//   Motion/Motion Instance <-> CX2020 (EtherCAT)/Term 1 (EK1200)/Term 2 (EK1122)/Rack#2B-01 Coupler (EK1100)/Rack#2B-09 ENC_RxG_XG (EL5042)
//     PlcTask Inputs/GVL_Main.M10.nRawEncoderULINT <-> FB Inputs Channel 1 compact/Position
//     PlcTask Inputs/GVL_Main.M11.nRawEncoderULINT <-> FB Inputs Channel 2/Position
//   Motion/Motion Instance <-> CX2020 (EtherCAT)/Term 1 (EK1200)/Term 2 (EK1122)/Rack#2B-01 Coupler (EK1100)/Rack#2B-10 ENC_YG1_YG2 (EL5042)
//     PlcTask Inputs/GVL_Main.M7.nRawEncoderULINT <-> FB Inputs Channel 1/Position
//     PlcTask Inputs/GVL_Main.M8.nRawEncoderULINT <-> FB Inputs Channel 2/Position
//   Motion/Motion Instance <-> CX2020 (EtherCAT)/Term 1 (EK1200)/Term 2 (EK1122)/Rack#2B-01 Coupler (EK1100)/Rack#2B-11 ENC_YG3_X1PM (EL5042)
//     PlcTask Inputs/GVL_Main.M12.nRawEncoderULINT <-> FB Inputs Channel 2/Position
//     PlcTask Inputs/GVL_Main.M9.nRawEncoderULINT <-> FB Inputs Channel 1/Position
//   Motion/Motion Instance <-> CX2020 (EtherCAT)/Term 1 (EK1200)/Term 2 (EK1122)/Rack#2B-01 Coupler (EK1100)/Rack#2B-12 ENC_X2PM_RzPM (EL5042)
//     PlcTask Inputs/GVL_Main.M13.nRawEncoderULINT <-> FB Inputs Channel 1/Position
//     PlcTask Inputs/GVL_Main.M14.nRawEncoderULINT <-> FB Inputs Channel 2/Position
//   Motion/Motion Instance <-> CX2020 (EtherCAT)/Term 1 (EK1200)/Term 2 (EK1122)/Rack#2B-01 Coupler (EK1100)/Rack#2B-15 DR_YDF1 (EL7041-0052)
//     PlcTask Inputs/GVL_Main.M15.bLimitBackwardEnable <-> STM Status/Status/Digital input 2
//     PlcTask Inputs/GVL_Main.M15.bLimitForwardEnable <-> STM Status/Status/Digital input 1
//   Motion/Motion Instance <-> CX2020 (EtherCAT)/Term 1 (EK1200)/Term 2 (EK1122)/Rack#2B-01 Coupler (EK1100)/Rack#2B-16 DR_YDF2 (EL7041-0052)
//     PlcTask Inputs/GVL_Main.M16.bLimitBackwardEnable <-> STM Status/Status/Digital input 2
//     PlcTask Inputs/GVL_Main.M16.bLimitForwardEnable <-> STM Status/Status/Digital input 1
//   Motion/Motion Instance <-> CX2020 (EtherCAT)/Term 1 (EK1200)/Term 2 (EK1122)/Rack#2B-01 Coupler (EK1100)/Rack#2B-18 MB_ZF (EL2602)
//     PlcTask Outputs/GVL_Main.M27.bBrakeRelease <-> Channel 1/Output
//   Motion/Motion Instance <-> CX2020 (EtherCAT)/Term 1 (EK1200)/Term 2 (EK1122)/Rack#2B-01 Coupler (EK1100)/Rack#2B-19 DR_YDF3 (EL7041-0052)
//     PlcTask Inputs/GVL_Main.M17.bLimitBackwardEnable <-> STM Status/Status/Digital input 2
//     PlcTask Inputs/GVL_Main.M17.bLimitForwardEnable <-> STM Status/Status/Digital input 1
//   Motion/Motion Instance <-> CX2020 (EtherCAT)/Term 1 (EK1200)/Term 2 (EK1122)/Rack#2D LinearGaugeAmp (SC-HG1-ETC)
//     PlcTask Inputs/GVL_Sensor.stHDF.iRawCnts <-> Process Data(In)  TxPDO-Map/Response Data Unit4
//     PlcTask Inputs/GVL_Sensor.stYDF1.iRawCnts <-> Process Data(In)  TxPDO-Map/Response Data Unit1
//     PlcTask Inputs/GVL_Sensor.stYDF2.iRawCnts <-> Process Data(In)  TxPDO-Map/Response Data Unit2
//     PlcTask Inputs/GVL_Sensor.stYDF3.iRawCnts <-> Process Data(In)  TxPDO-Map/Response Data Unit3
//     PlcTask Outputs/PRG_Sensor.bSensorHeadNormalValueMode <-> Process Data(Out) RxPDO-Map/Normal Value Mode
//     PlcTask Outputs/PRG_Sensor.bSensorHeadValueMode <-> Process Data(Out) RxPDO-Map/Head Value Mode
//   Motion/Motion Instance <-> NC-Task 1 SAF/Axes/RxG
//     PlcTask Inputs/GVL_Main.M10.Axis.NcToPlc <-> Outputs/ToPlc
//     PlcTask Outputs/GVL_Main.M10.Axis.PlcToNc <-> Inputs/FromPlc
//   Motion/Motion Instance <-> NC-Task 1 SAF/Axes/RyDC
//     PlcTask Inputs/GVL_Main.M23.Axis.NcToPlc <-> Outputs/ToPlc
//     PlcTask Outputs/GVL_Main.M23.Axis.PlcToNc <-> Inputs/FromPlc
//   Motion/Motion Instance <-> NC-Task 1 SAF/Axes/RzPM
//     PlcTask Inputs/GVL_Main.M14.Axis.NcToPlc <-> Outputs/ToPlc
//     PlcTask Outputs/GVL_Main.M14.Axis.PlcToNc <-> Inputs/FromPlc
//   Motion/Motion Instance <-> NC-Task 1 SAF/Axes/Stepper
//     PlcTask Inputs/GVL_Main.M2.Axis.NcToPlc <-> Outputs/ToPlc
//     PlcTask Outputs/GVL_Main.M2.Axis.PlcToNc <-> Inputs/FromPlc
//   Motion/Motion Instance <-> NC-Task 1 SAF/Axes/XDC
//     PlcTask Inputs/GVL_Main.M22.Axis.NcToPlc <-> Outputs/ToPlc
//     PlcTask Outputs/GVL_Main.M22.Axis.PlcToNc <-> Inputs/FromPlc
//   Motion/Motion Instance <-> NC-Task 1 SAF/Axes/XG
//     PlcTask Inputs/GVL_Main.M11.Axis.NcToPlc <-> Outputs/ToPlc
//     PlcTask Outputs/GVL_Main.M11.Axis.PlcToNc <-> Inputs/FromPlc
//   Motion/Motion Instance <-> NC-Task 1 SAF/Axes/XPM1
//     PlcTask Inputs/GVL_Main.M12.Axis.NcToPlc <-> Outputs/ToPlc
//     PlcTask Outputs/GVL_Main.M12.Axis.PlcToNc <-> Inputs/FromPlc
//   Motion/Motion Instance <-> NC-Task 1 SAF/Axes/XPM2
//     PlcTask Inputs/GVL_Main.M13.Axis.NcToPlc <-> Outputs/ToPlc
//     PlcTask Outputs/GVL_Main.M13.Axis.PlcToNc <-> Inputs/FromPlc
//   Motion/Motion Instance <-> NC-Task 1 SAF/Axes/XS1
//     PlcTask Inputs/GVL_Main.M3.Axis.NcToPlc <-> Outputs/ToPlc
//     PlcTask Outputs/GVL_Main.M3.Axis.PlcToNc <-> Inputs/FromPlc
//   Motion/Motion Instance <-> NC-Task 1 SAF/Axes/XS2
//     PlcTask Inputs/GVL_Main.M4.Axis.NcToPlc <-> Outputs/ToPlc
//     PlcTask Outputs/GVL_Main.M4.Axis.PlcToNc <-> Inputs/FromPlc
//   Motion/Motion Instance <-> NC-Task 1 SAF/Axes/XSDC1
//     PlcTask Inputs/GVL_Main.M18.Axis.NcToPlc <-> Outputs/ToPlc
//     PlcTask Outputs/GVL_Main.M18.Axis.PlcToNc <-> Inputs/FromPlc
//   Motion/Motion Instance <-> NC-Task 1 SAF/Axes/XSDC2
//     PlcTask Inputs/GVL_Main.M19.Axis.NcToPlc <-> Outputs/ToPlc
//     PlcTask Outputs/GVL_Main.M19.Axis.PlcToNc <-> Inputs/FromPlc
//   Motion/Motion Instance <-> NC-Task 1 SAF/Axes/YDF1
//     PlcTask Inputs/GVL_Main.M15.Axis.NcToPlc <-> Outputs/ToPlc
//     PlcTask Outputs/GVL_Main.M15.Axis.PlcToNc <-> Inputs/FromPlc
//   Motion/Motion Instance <-> NC-Task 1 SAF/Axes/YDF2
//     PlcTask Inputs/GVL_Main.M16.Axis.NcToPlc <-> Outputs/ToPlc
//     PlcTask Outputs/GVL_Main.M16.Axis.PlcToNc <-> Inputs/FromPlc
//   Motion/Motion Instance <-> NC-Task 1 SAF/Axes/YDF3
//     PlcTask Inputs/GVL_Main.M17.Axis.NcToPlc <-> Outputs/ToPlc
//     PlcTask Outputs/GVL_Main.M17.Axis.PlcToNc <-> Inputs/FromPlc
//   Motion/Motion Instance <-> NC-Task 1 SAF/Axes/YF1
//     PlcTask Inputs/GVL_Main.M25.Axis.NcToPlc <-> Outputs/ToPlc
//     PlcTask Outputs/GVL_Main.M25.Axis.PlcToNc <-> Inputs/FromPlc
//   Motion/Motion Instance <-> NC-Task 1 SAF/Axes/YF2
//     PlcTask Inputs/GVL_Main.M26.Axis.NcToPlc <-> Outputs/ToPlc
//     PlcTask Outputs/GVL_Main.M26.Axis.PlcToNc <-> Inputs/FromPlc
//   Motion/Motion Instance <-> NC-Task 1 SAF/Axes/YG1
//     PlcTask Inputs/GVL_Main.M7.Axis.NcToPlc <-> Outputs/ToPlc
//     PlcTask Outputs/GVL_Main.M7.Axis.PlcToNc <-> Inputs/FromPlc
//   Motion/Motion Instance <-> NC-Task 1 SAF/Axes/YG2
//     PlcTask Inputs/GVL_Main.M8.Axis.NcToPlc <-> Outputs/ToPlc
//     PlcTask Outputs/GVL_Main.M8.Axis.PlcToNc <-> Inputs/FromPlc
//   Motion/Motion Instance <-> NC-Task 1 SAF/Axes/YG3
//     PlcTask Inputs/GVL_Main.M9.Axis.NcToPlc <-> Outputs/ToPlc
//     PlcTask Outputs/GVL_Main.M9.Axis.PlcToNc <-> Inputs/FromPlc
//   Motion/Motion Instance <-> NC-Task 1 SAF/Axes/YS1
//     PlcTask Inputs/GVL_Main.M5.Axis.NcToPlc <-> Outputs/ToPlc
//     PlcTask Outputs/GVL_Main.M5.Axis.PlcToNc <-> Inputs/FromPlc
//   Motion/Motion Instance <-> NC-Task 1 SAF/Axes/YS2
//     PlcTask Inputs/GVL_Main.M6.Axis.NcToPlc <-> Outputs/ToPlc
//     PlcTask Outputs/GVL_Main.M6.Axis.PlcToNc <-> Inputs/FromPlc
//   Motion/Motion Instance <-> NC-Task 1 SAF/Axes/YSDC1
//     PlcTask Inputs/GVL_Main.M20.Axis.NcToPlc <-> Outputs/ToPlc
//     PlcTask Outputs/GVL_Main.M20.Axis.PlcToNc <-> Inputs/FromPlc
//   Motion/Motion Instance <-> NC-Task 1 SAF/Axes/YSDC2
//     PlcTask Inputs/GVL_Main.M21.Axis.NcToPlc <-> Outputs/ToPlc
//     PlcTask Outputs/GVL_Main.M21.Axis.PlcToNc <-> Inputs/FromPlc
//   Motion/Motion Instance <-> NC-Task 1 SAF/Axes/ZDC
//     PlcTask Inputs/GVL_Main.M24.Axis.NcToPlc <-> Outputs/ToPlc
//     PlcTask Outputs/GVL_Main.M24.Axis.PlcToNc <-> Inputs/FromPlc
//   Motion/Motion Instance <-> NC-Task 1 SAF/Axes/ZF
//     PlcTask Inputs/GVL_Main.M27.Axis.NcToPlc <-> Outputs/ToPlc
//     PlcTask Outputs/GVL_Main.M27.Axis.PlcToNc <-> Inputs/FromPlc

CONFIGURATION Motion
    RESOURCE PLC ON TwinCAT3
        TASK PlcTask(INTERVAL := T#10ms, PRIORITY := 20);
        PROGRAM PRG1_MAIN_PlcTask WITH PlcTask : PRG1_MAIN_PlcTask;
    END_RESOURCE
END_CONFIGURATION

// ---- DUTs/DUT_SensorHGS.TcDUT
TYPE DUT_SensorHGS:
STRUCT 
	fCntsInEGU:			REAL;
	sEGU:				STRING;
	sName:				STRING;
	fValue:				REAL;
	iRawCnts AT %I*:	DINT;
	iOffset:			DINT;
	q_iRawCnts AT %I*:	UINT;
END_STRUCT
END_TYPE

// ---- GVLs/GVL_Main.TcGVL
{attribute 'qualified_only'}
VAR_GLOBAL
	bResetIClk: BOOL;
	{attribute 'TcLinkTo' := 'TIIB[Rack#1A-02 SFIN (EL1918)]^StandardInputs^Standard Out Var 18'}
	bESTOP AT %I*: BOOL;
	
	{attribute 'TcLinkTo' := 'TIIB[Rack#2B-05 SV_AIR (EL2004)]^Channel 1^Output'}
	bOpenSV1 AT %Q*: BOOL;
	{attribute 'TcLinkTo' := 'TIIB[Rack#2B-05 SV_AIR (EL2004)]^Channel 2^Output'}
	bOpenSV2 AT %Q*: BOOL;
	
	{attribute 'TcLinkTo' := 'TIIB[Rack#1C_ServoDR (NCR-HD Series)]^260th receive PDO Mapping^Positive torque limit value'}
	iServoTorqueLimitPositive AT %Q*: UINT;
	
	{attribute 'TcLinkTo' := 'TIIB[Rack#1C_ServoDR (NCR-HD Series)]^260th receive PDO Mapping^Negative torque limit value'}
	iServoTorqueLimitNegative AT %Q*: UINT;

	// 2Theta Servo
	M1: DUT_MotionStage;
	
	// 2Theta Stepper
	{attribute 'TcLinkTo' := '	.bLimitForwardEnable  	:= TIIB[Rack#1A-04 DR_2Th (EL7047)]^STM Status^Status^Digital input 1;
								.bLimitBackwardEnable 	:= TIIB[Rack#1A-04 DR_2Th (EL7047)]^STM Status^Status^Digital input 2;
								.nRawEncoderULINT     	:= TIIB[Rack#1A-06 ENC_2Th (EL5042)]^FB Inputs Channel 1^Position;
								.bBrakeRelease			:= TIIB[Rack#1A-05 MB_2Th (EL2602)]^Channel 1^Output
	'}
	M2: DUT_MotionStage;
	
	// XS1
	{attribute 'TcLinkTo' := '	.bLimitForwardEnable  	:= TIIB[Rack#2A-03 DR_XS1 (EL7041-0052)]^STM Status^Status^Digital input 1;
								.bLimitBackwardEnable 	:= TIIB[Rack#2A-03 DR_XS1 (EL7041-0052)]^STM Status^Status^Digital input 2;
								.nRawEncoderULINT     	:= TIIB[Rack#2B-07 ENC_X1_X2 (EL5042)]^FB Inputs Channel 1^Position
	'}
    M3: DUT_MotionStage;
	
	// XS2
	{attribute 'TcLinkTo' := '	.bLimitForwardEnable  	:= TIIB[Rack#2A-04 DR_XS2 (EL7041-0052)]^STM Status^Status^Digital input 1;
								.bLimitBackwardEnable 	:= TIIB[Rack#2A-04 DR_XS2 (EL7041-0052)]^STM Status^Status^Digital input 2;
								.nRawEncoderULINT     	:= TIIB[Rack#2B-07 ENC_X1_X2 (EL5042)]^FB Inputs Channel 2^Position
	'}
    M4: DUT_MotionStage;
	
	// YS1
	{attribute 'TcLinkTo' := '	.bLimitForwardEnable  	:= TIIB[Rack#2A-05 DR_YS1 (EL7041-0052)]^STM Status^Status^Digital input 1;
								.bLimitBackwardEnable 	:= TIIB[Rack#2A-05 DR_YS1 (EL7041-0052)]^STM Status^Status^Digital input 2;
								.nRawEncoderULINT     	:= TIIB[Rack#2B-08 ENC_Y1_Y2 (EL5042)]^FB Inputs Channel 1^Position
	'}
    M5: DUT_MotionStage;
	
	// YS2
	{attribute 'TcLinkTo' := '	.bLimitForwardEnable  	:= TIIB[Rack#2A-06 DR_YS2 (EL7041-0052)]^STM Status^Status^Digital input 1;
								.bLimitBackwardEnable 	:= TIIB[Rack#2A-06 DR_YS2 (EL7041-0052)]^STM Status^Status^Digital input 2;
								.nRawEncoderULINT     	:= TIIB[Rack#2B-08 ENC_Y1_Y2 (EL5042)]^FB Inputs Channel 1^Position
	'}
    M6: DUT_MotionStage;
	
	// YG1
    {attribute 'TcLinkTo' := '	.bLimitForwardEnable	:= TIIB[Rack#2A-10 DR_YG1 (EL7041-0052)]^STM Status^Status^Digital input 1;
								.bLimitBackwardEnable	:= TIIB[Rack#2A-10 DR_YG1 (EL7041-0052)]^STM Status^Status^Digital input 2;
								.nRawEncoderULINT		:= TIIB[Rack#2B-10 ENC_YG1_YG2 (EL5042)]^FB Inputs Channel 1^Position
	'}
	M7: DUT_MotionStage;
	
	// YG2
    {attribute 'TcLinkTo' := '	.bLimitForwardEnable	:= TIIB[Rack#2A-11 DR_YG2 (EL7041-0052)]^STM Status^Status^Digital input 1;
								.bLimitBackwardEnable	:= TIIB[Rack#2A-11 DR_YG2 (EL7041-0052)]^STM Status^Status^Digital input 2;
								.nRawEncoderULINT		:= TIIB[Rack#2B-10 ENC_YG1_YG2 (EL5042)]^FB Inputs Channel 2^Position
	'}
    M8: DUT_MotionStage;
	
	// YG3
    {attribute 'TcLinkTo' := '	.bLimitForwardEnable	:= TIIB[Rack#2A-12 DR_YG3 (EL7041-0052)]^STM Status^Status^Digital input 1;
								.bLimitBackwardEnable	:= TIIB[Rack#2A-12 DR_YG3 (EL7041-0052)]^STM Status^Status^Digital input 2;
								.nRawEncoderULINT		:= TIIB[Rack#2B-11 ENC_YG3_X1PM (EL5042)]^FB Inputs Channel 1^Position
	'}
    M9: DUT_MotionStage;
	
	
	// RxG
    {attribute 'TcLinkTo' := '	.bLimitForwardEnable	:= TIIB[Rack#2A-08 DR_RxG (EL7041-0052)]^STM Status^Status^Digital input 1;
								.bLimitBackwardEnable	:= TIIB[Rack#2A-08 DR_RxG (EL7041-0052)]^STM Status^Status^Digital input 2;
								.nRawEncoderULINT		:= TIIB[Rack#2B-09 ENC_RxG_XG (EL5042)]^FB Inputs Channel 1 compact^Position
	'}
    M10: DUT_MotionStage;
	
	// XG
    {attribute 'TcLinkTo' := '	.bLimitForwardEnable	:= TIIB[Rack#2A-09 DR_XG (EL7041-0052)]^STM Status^Status^Digital input 1;
								.bLimitBackwardEnable	:= TIIB[Rack#2A-09 DR_XG (EL7041-0052)]^STM Status^Status^Digital input 2;
								.nRawEncoderULINT		:= TIIB[Rack#2B-09 ENC_RxG_XG (EL5042)]^FB Inputs Channel 2^Position
	'}
    M11: DUT_MotionStage;
	
	// XPM1
    {attribute 'TcLinkTo' := '	.bLimitForwardEnable	:= TIIB[Rack#2A-14 DR_XPM1 (EL7041-0052)]^STM Status^Status^Digital input 1;
								.bLimitBackwardEnable	:= TIIB[Rack#2A-14 DR_XPM1 (EL7041-0052)]^STM Status^Status^Digital input 2;
								.nRawEncoderULINT		:= TIIB[Rack#2B-11 ENC_YG3_X1PM (EL5042)]^FB Inputs Channel 2^Position
	'}
    M12: DUT_MotionStage;
	
	// XPM2
    {attribute 'TcLinkTo' := '	.bLimitForwardEnable	:= TIIB[Rack#2A-15 DR_XPM2 (EL7041-0052)]^STM Status^Status^Digital input 1;
								.bLimitBackwardEnable	:= TIIB[Rack#2A-15 DR_XPM2 (EL7041-0052)]^STM Status^Status^Digital input 2;
								.nRawEncoderULINT		:= TIIB[Rack#2B-12 ENC_X2PM_RzPM (EL5042)]^FB Inputs Channel 1^Position
	'}
	M13: DUT_MotionStage;
	
	// RzPM
    {attribute 'TcLinkTo' := '	.bLimitForwardEnable	:= TIIB[Rack#2A-16 DR_RzPM (EL7041-0052)]^STM Status^Status^Digital input 1;
								.bLimitBackwardEnable	:= TIIB[Rack#2A-16 DR_RzPM (EL7041-0052)]^STM Status^Status^Digital input 2;
								.nRawEncoderULINT		:= TIIB[Rack#2B-12 ENC_X2PM_RzPM (EL5042)]^FB Inputs Channel 2^Position
	'}
    M14: DUT_MotionStage;

	// YDF1
	{attribute 'TcLinkTo' := '	.bLimitForwardEnable  	:= TIIB[Rack#2B-15 DR_YDF1 (EL7041-0052)]^STM Status^Status^Digital input 1;
								.bLimitBackwardEnable 	:= TIIB[Rack#2B-15 DR_YDF1 (EL7041-0052)]^STM Status^Status^Digital input 2
	'}
    M15: DUT_MotionStage;
	
	// YDF2
	{attribute 'TcLinkTo' := '	.bLimitForwardEnable  	:= TIIB[Rack#2B-16 DR_YDF2 (EL7041-0052)]^STM Status^Status^Digital input 1;
								.bLimitBackwardEnable 	:= TIIB[Rack#2B-16 DR_YDF2 (EL7041-0052)]^STM Status^Status^Digital input 2
	'}
    M16: DUT_MotionStage;
	
	// YDF3
	{attribute 'TcLinkTo' := '	.bLimitForwardEnable  	:= TIIB[Rack#2B-19 DR_YDF3 (EL7041-0052)]^STM Status^Status^Digital input 1;
								.bLimitBackwardEnable 	:= TIIB[Rack#2B-19 DR_YDF3 (EL7041-0052)]^STM Status^Status^Digital input 2
	'}
    M17: DUT_MotionStage;
	
	// XSDC1
	{attribute 'TcLinkTo' := '	.bLimitForwardEnable  	:= TIIB[BOX-09 DR_XSDC1 (EL7041-0052)]^STM Status^Status^Digital input 1;
								.bLimitBackwardEnable 	:= TIIB[BOX-09 DR_XSDC1 (EL7041-0052)]^STM Status^Status^Digital input 2;
								.nRawEncoderULINT     	:= TIIB[BOX-03 ENC_X1_X2 (EL5042)]^FB Inputs Channel 1^Position
	'}
    M18: DUT_MotionStage;
	
	// XSDC2
	{attribute 'TcLinkTo' := '	.bLimitForwardEnable	:= TIIB[BOX-10 DR_XSDC2 (EL7041-0052)]^STM Status^Status^Digital input 1;
								.bLimitBackwardEnable 	:= TIIB[BOX-10 DR_XSDC2 (EL7041-0052)]^STM Status^Status^Digital input 2;
								.nRawEncoderULINT     	:= TIIB[BOX-03 ENC_X1_X2 (EL5042)]^FB Inputs Channel 2^Position
	'}
    M19: DUT_MotionStage;
	
	// YSDC1
	{attribute 'TcLinkTo' := '	.bLimitForwardEnable	:= TIIB[BOX-11 DR_YSDC1 (EL7041-0052)]^STM Status^Status^Digital input 1;
								.bLimitBackwardEnable 	:= TIIB[BOX-11 DR_YSDC1 (EL7041-0052)]^STM Status^Status^Digital input 2;
								.nRawEncoderULINT     	:= TIIB[BOX-04 ENC_Y1_Y2 (EL5042)]^FB Inputs Channel 1^Position
	'}
    M20: DUT_MotionStage;
	
	// YSDC2
	{attribute 'TcLinkTo' := '	.bLimitForwardEnable	:= TIIB[BOX-12 DR_YSDC2 (EL7041-0052)]^STM Status^Status^Digital input 1;
								.bLimitBackwardEnable 	:= TIIB[BOX-12 DR_YSDC2 (EL7041-0052)]^STM Status^Status^Digital input 2;
								.nRawEncoderULINT     	:= TIIB[BOX-04 ENC_Y1_Y2 (EL5042)]^FB Inputs Channel 1^Position
	'}
    M21: DUT_MotionStage;

	// XDC
	{attribute 'TcLinkTo' := '	.bLimitForwardEnable  	:= TIIB[BOX-14 DR_XDC (EL7041-0052)]^STM Status^Status^Digital input 1;
								.bLimitBackwardEnable 	:= TIIB[BOX-14 DR_XDC (EL7041-0052)]^STM Status^Status^Digital input 2;
								.nRawEncoderULINT     	:= TIIB[BOX-05 ENC_XDC_RyDC (EL5042)]^FB Inputs Channel 1^Position
	'}
    M22: DUT_MotionStage;
	
	// RyDC
	{attribute 'TcLinkTo' := '	.bLimitForwardEnable	:= TIIB[BOX-15 DR_RyDC (EL7041-0052)]^STM Status^Status^Digital input 1;
								.bLimitBackwardEnable	:= TIIB[BOX-15 DR_RyDC (EL7041-0052)]^STM Status^Status^Digital input 2;
								.nRawEncoderULINT		:= TIIB[BOX-05 ENC_XDC_RyDC (EL5042)]^FB Inputs Channel 2^Position
	'}
    M23: DUT_MotionStage;
	
	// ZDC
	{attribute 'TcLinkTo' := '	.bLimitForwardEnable	:= TIIB[BOX-16 DR_ZDC (EL7041-0052)]^STM Status^Status^Digital input 1;
								.bLimitBackwardEnable	:= TIIB[BOX-16 DR_ZDC (EL7041-0052)]^STM Status^Status^Digital input 2;
								.nRawEncoderULINT		:= TIIB[BOX-06 ENC_ZDC_YF1 (EL5042)]^FB Inputs Channel 1^Position
	'}
    M24: DUT_MotionStage;

	// YF1
	{attribute 'TcLinkTo' := '	.bLimitForwardEnable	:= TIIB[Rack#1A-02 SFIN (EL1918)]^StandardInputs^Standard Out Var 10;
								.bLimitBackwardEnable 	:= TIIB[Rack#1A-02 SFIN (EL1918)]^StandardInputs^Standard Out Var 11;
								.nRawEncoderULINT     	:= TIIB[BOX-06 ENC_ZDC_YF1 (EL5042)]^FB Inputs Channel 2^Position;
								.bBrakeRelease        	:= TIIB[BOX-19 MB_YF1_YF2 (EL2602)]^Channel 1^Output
	'}
    M25: DUT_MotionStage;
	
	// YF2
	{attribute 'TcLinkTo' := '	.bLimitForwardEnable	:= TIIB[Rack#1A-02 SFIN (EL1918)]^StandardInputs^Standard Out Var 12;
								.bLimitBackwardEnable	:= TIIB[Rack#1A-02 SFIN (EL1918)]^StandardInputs^Standard Out Var 13;
								.nRawEncoderULINT     	:= TIIB[BOX-07 ENC_YF2_ZF (EL5042)]^FB Inputs Channel 1^Position;
								.bBrakeRelease			:= TIIB[BOX-19 MB_YF1_YF2 (EL2602)]^Channel 2^Output
	'}
	M26: DUT_MotionStage;
	
	// ZF
	{attribute 'TcLinkTo' := '	.bLimitForwardEnable	:= TIIB[Rack#1A-02 SFIN (EL1918)]^StandardInputs^Standard Out Var 14;
								.bLimitBackwardEnable	:= TIIB[Rack#1A-02 SFIN (EL1918)]^StandardInputs^Standard Out Var 15;
								.nRawEncoderULINT		:= TIIB[BOX-07 ENC_YF2_ZF (EL5042)]^FB Inputs Channel 2^Position;
								.bBrakeRelease			:= TIIB[Rack#2B-18 MB_ZF (EL2602)]^Channel 1^Output
	'}
	M27: DUT_MotionStage;
	
	
END_VAR

// ---- GVLs/GVL_PMPS.TcGVL
{attribute 'qualified_only'}
VAR_GLOBAL
	fbArbiter: FB_Arbiter(1);
	io_fbFFHWO: FB_HardwareFFOutput;
END_VAR

// ---- POUs/PRG1_MAIN_PlcTask.TcPOU
PROGRAM PRG1_MAIN_PlcTask
VAR	
    {attribute 'TcLinkTo' := 'TIIB[Rack#1A-01 Coupler (EK1100)]^Rack#1A-02 SFIN (EL1918)^StandardOutputs^Standard In Var 2'}
	bEnaIclk AT %Q*: BOOL := TRUE;
	
    {attribute 'TcLinkTo' := 'TIIB[Rack#1A-01 Coupler (EK1100)]^Rack#1A-02 SFIN (EL1918)^StandardOutputs^Standard In Var 1'}
	bEnaIclkErrAck AT %Q*: BOOL := FALSE;
	
    {attribute 'TcLinkTo' := 'TIIB[Rack#1A-01 Coupler (EK1100)]^Rack#1A-02 SFIN (EL1918)^StandardOutputs^Standard In Var 9'}
	bEnaIclkRestartESTOP AT %Q*: BOOL := FALSE;
	
	fbPower_AxisM11: MC_Power;
	fbPower_AxisM12: MC_Power;
	fbPower_AxisM13: MC_Power;
	fbPower_AxisM14: MC_Power;
END_VAR

ACT_ESTOP();

PRG_2Theta();
PRG_DET_ARM();
PRG_DET_CHAMBER();
PRG_DET_SLIT();
PRG_DET_FRAME();
PRG_OPT_SLITS();
PRG_OPT_YG();
PRG_OPT_XPM();
PRG_OPT();
PRG_Sensor();

ACTION ACT_ESTOP:

IF bEnaIclkErrAck THEN
	bEnaIclkErrAck := FALSE;
END_IF
IF bEnaIclkRestartESTOP THEN
	bEnaIclkRestartESTOP := FALSE;
END_IF

// When user push the ESTOPs
IF NOT GVL_Main.bESTOP THEN
	
	GVL_Main.bOpenSV1 := FALSE;
	GVL_Main.bOpenSV2 := FALSE;

	GVL_Main.M1.bEnable := FALSE;
	GVL_Main.M2.bEnable := FALSE;
	GVL_Main.M3.bEnable := FALSE;
	GVL_Main.M4.bEnable := FALSE;
	GVL_Main.M5.bEnable := FALSE;
	GVL_Main.M6.bEnable := FALSE;
	GVL_Main.M7.bEnable := FALSE;
	GVL_Main.M8.bEnable := FALSE;
	GVL_Main.M9.bEnable := FALSE;
	GVL_Main.M10.bEnable := FALSE;
	GVL_Main.M11.bEnable := FALSE;
	GVL_Main.M12.bEnable := FALSE;
	GVL_Main.M13.bEnable := FALSE;
	GVL_Main.M14.bEnable := FALSE;
	GVL_Main.M15.bEnable := FALSE;
	GVL_Main.M16.bEnable := FALSE;
	GVL_Main.M17.bEnable := FALSE;
	GVL_Main.M18.bEnable := FALSE;
	GVL_Main.M19.bEnable := FALSE;
	GVL_Main.M20.bEnable := FALSE;
	GVL_Main.M21.bEnable := FALSE;
	GVL_Main.M22.bEnable := FALSE;
	GVL_Main.M23.bEnable := FALSE;
	GVL_Main.M24.bEnable := FALSE;
	GVL_Main.M25.bEnable := FALSE;
	GVL_Main.M26.bEnable := FALSE;
	GVL_Main.M27.bEnable := FALSE;
END_IF


// Disable M1(Servo) and M2(Stepper) if the frame is landing...
IF NOT GVL_Sensor.bFloating THEN
	GVL_Main.M1.bEnable := FALSE;
	GVL_Main.M2.bEnable := FALSE;
END_IF
	

// When user requests to reset ESTOP.
IF GVL_Main.bResetIclk THEN
	GVL_Main.bResetIclk := FALSE;	
	bEnaIclkErrAck := TRUE;
	bEnaIclkRestartESTOP := TRUE;
END_IF
END_ACTION

END_PROGRAM

// ---- POUs/PRG_2Theta.TcPOU
PROGRAM PRG_2Theta
VAR
	bInit: BOOL := TRUE;
	fbPower_AxisM1:  MC_Power;
	fbPower_AxisM2:  MC_Power;
	fb2ThetaStepper : FB_MotionStage;
	fb2ThetaServo : FB_MotionStage;
	bMoveOk: BOOL;
	
	
	
	fThresholdPS1: REAL := 0.15;
	fThresholdPS2: REAL;
	fThresholdPS3: REAL;
 
END_VAR

IF binit THEN
	bInit := FALSE;
	
	// Servo
	GVL_Main.M1.nBrakeMode := ENUM_StageBrakeMode.NO_BRAKE;
	GVL_Main.M1.bHardwareEnable := TRUE;
	GVL_Main.M1.bPowerSelf := FALSE;
	
	// Set torque output limit (unit: 0.1%)
	GVL_Main.iServoTorqueLimitPositive := 1500; // 1500*0.1% = 150%
	GVL_Main.iServoTorqueLimitNegative := 1500;
	
	// Stepper
	GVL_Main.M2.nBrakeMode := ENUM_StageBrakeMode.IF_MOVING;
	GVL_Main.M2.bHardwareEnable := TRUE;
	GVL_Main.M2.bPowerSelf := FALSE;
END_IF;

ACT_Servo();
ACT_Stepper();

ACTION ACT_Servo:
fb2ThetaServo(stMotionStage:=GVL_Main.M1);

GVL_Main.M1.bPowerSelf := FALSE;

GVL_Main.M1.bAllEnable := 		GVL_Main.M1.bEnable
							AND GVL_Main.bESTOP // ESTOP
							AND	GVL_Sensor.stPS1.fValue > fThresholdPS1
							AND GVL_Sensor.stPS2.fValue > fThresholdPS2
							AND GVL_Sensor.stPS3.fValue > fThresholdPS3; // Compressed-air pressure
GVL_Main.M1.bAllForwardEnable  := GVL_Main.M1.bLimitForwardEnable  AND GVL_Main.bESTOP;
GVL_Main.M1.bAllBackwardEnable := GVL_Main.M1.bLimitBackwardEnable AND GVL_Main.bESTOP;

fbPower_AxisM1(
	Axis:= GVL_Main.M1.Axis,
	Enable := GVL_Main.M1.bAllEnable,
	Enable_Positive:= GVL_Main.M1.bAllForwardEnable,
	Enable_Negative:= GVL_Main.M1.bAllBackwardEnable,
	Override:= 100
);
END_ACTION

ACTION ACT_Stepper:
fb2ThetaStepper(stMotionStage:=GVL_Main.M2);

GVL_Main.M2.bPowerSelf := FALSE;

GVL_Main.M2.bAllEnable := 		GVL_Main.M2.bEnable
							AND GVL_Main.bESTOP // ESTOP
							AND	GVL_Sensor.stPS1.fValue > fThresholdPS1
							AND GVL_Sensor.stPS2.fValue > fThresholdPS2
							AND GVL_Sensor.stPS3.fValue > fThresholdPS3; // Compressed-air pressure
GVL_Main.M2.bAllForwardEnable  := GVL_Main.M2.bLimitForwardEnable  AND GVL_Main.bESTOP;
GVL_Main.M2.bAllBackwardEnable := GVL_Main.M2.bLimitBackwardEnable AND GVL_Main.bESTOP;

fbPower_AxisM2(
	Axis:= GVL_Main.M2.Axis,
	Enable := GVL_Main.M2.bAllEnable,
	Enable_Positive:= GVL_Main.M2.bAllForwardEnable,
	Enable_Negative:= GVL_Main.M2.bAllBackwardEnable,
	Override:= 100
);
END_ACTION

END_PROGRAM

// ---- POUs/PRG_DET_ARM.TcPOU
PROGRAM PRG_DET_ARM
VAR
	bInit: BOOL := TRUE;
	bExecuteCouple: BOOL := FALSE;
	bExecuteDecouple: BOOL := FALSE;
	
	fbMotionYF1: FB_MotionStage;
	fbMotionYF2: FB_MotionStage;
	fbMotionZF: FB_MotionStage;
	fbAutoCoupling: FB_GantryAutoCoupling;
	
	{attribute 'TcLinkTo' := '	.Count := TIIB[BOX-06 ENC_ZDC_YF1 (EL5042)]^FB Inputs Channel 2^Position'}
	stRenishawAbsEncMaster: ST_RenishawAbsEnc;
	{attribute 'TcLinkTo' := '	.Count := TIIB[BOX-07 ENC_YF2_ZF (EL5042)]^FB Inputs Channel 1^Position'}
	stRenishawAbsEncSlave: ST_RenishawAbsEnc;

	(*
	fbPower_AxisM25: MC_POWER;
	fbPower_AxisM26: MC_POWER;
	fbPower_AxisM27: MC_POWER;
	
	tonBrakeRlease_M25, tonBrakeRlease_M26, tonBrakeRlease_M27: TON;
	// *)
END_VAR

IF bInit THEN
	bInit := FALSE;
	bExecuteCouple := TRUE;
	
	GVL_Main.M25.nBrakeMode := ENUM_StageBrakeMode.IF_MOVING;
	GVL_Main.M25.bHardwareEnable := TRUE;
	GVL_Main.M25.bPowerSelf := TRUE;
	GVL_Main.M26.nBrakeMode := ENUM_StageBrakeMode.IF_MOVING;
	GVL_Main.M26.bHardwareEnable := TRUE;
	GVL_Main.M26.bPowerSelf := TRUE;
	GVL_Main.M27.nBrakeMode := ENUM_StageBrakeMode.IF_ENABLED;
	GVL_Main.M27.bHardwareEnable := TRUE;
	GVL_Main.M27.bPowerSelf := TRUE;
END_IF

stRenishawAbsEncMaster.Ref := 15370335;
stRenishawAbsEncSlave.Ref := 15347257;

// AutoCoupling
fbAutoCoupling(	nGantryTol 			:= 200000, // 50nm/count
				Master				:= GVL_Main.M25,
				MasterEnc			:= stRenishawAbsEncMaster,
				Slave				:= GVL_Main.M26,
				SlaveEnc			:= stRenishawAbsEncSlave,
				bExecuteCouple 		:= bExecuteCouple,
				bExecuteDecouple 	:= bExecuteDecouple,
);

GVL_Main.M25.bAllEnable := GVL_Main.M25.bEnable AND GVL_Main.bESTOP;
GVL_Main.M26.bAllEnable := GVL_Main.M26.bEnable AND GVL_Main.bESTOP;
GVL_Main.M27.bAllEnable := GVL_Main.M27.bEnable AND GVL_Main.bESTOP;

// Call Motion FB instance
fbMotionYF1(stMotionStage:=GVL_Main.M25);
fbMotionYF2(stMotionStage:=GVL_Main.M26);
fbMotionZF(stMotionStage:=GVL_Main.M27);

(* For test
// Release brake if axis is enabled.
tonBrakeRlease_M25(
	IN:=(GVL_Main.M25.bEnable OR GVL_Main.M25.bAllEnable) AND NOT GVL_Main.M25.Axis.Status.DriveDeviceError,
	PT:=T#1s,
	Q=>GVL_Main.M25.bBrakeRelease
);
tonBrakeRlease_M26(
	IN:=(GVL_Main.M26.bEnable OR GVL_Main.M26.bAllEnable) AND NOT GVL_Main.M26.Axis.Status.DriveDeviceError,
	PT:=T#1s,
	Q=>GVL_Main.M26.bBrakeRelease
);
tonBrakeRlease_M27(
	IN:=(GVL_Main.M27.bEnable OR GVL_Main.M27.bAllEnable) AND NOT GVL_Main.M27.Axis.Status.DriveDeviceError,
	PT:=T#1s,
	Q=>GVL_Main.M27.bBrakeRelease
);
fbPower_AxisM25(
	Axis := GVL_Main.M25.Axis,
	Enable := GVL_Main.M25.bEnable AND GVL_Main.bESTOP,
	Enable_Positive := GVL_Main.M25.bLimitForwardEnable AND PLimFwd,
	Enable_Negative := GVL_Main.M25.bLimitBackwardEnable AND PLimBwd,
	Override := 100.000,
);
fbPower_AxisM26(
	Axis := GVL_Main.M26.Axis,
	Enable := GVL_Main.M26.bEnable AND GVL_Main.bESTOP,
	Enable_Positive := GVL_Main.M26.bLimitForwardEnable AND SLimFwd,
	Enable_Negative := GVL_Main.M26.bLimitBackwardEnable AND SLimBwd,
	Override := 100.000,
);
fbPower_AxisM27(
	Axis := GVL_Main.M27.Axis,
	Enable := GVL_Main.M27.bEnable AND GVL_Main.bESTOP,
	Enable_Positive := GVL_Main.M27.bLimitForwardEnable,
	Enable_Negative := GVL_Main.M27.bLimitBackwardEnable,
	Override := 100.000,
);


// *)

END_PROGRAM

// ---- POUs/PRG_DET_CHAMBER.TcPOU
PROGRAM PRG_DET_CHAMBER
VAR	
	bInit: BOOL := TRUE;
	fbMotionXDC: FB_MotionStage;
	fbMotionRyDC: FB_MotionStage;
	fbMotionZDC: FB_MotionStage;
END_VAR

// Det. Chmber
IF bInit THEN
	bInit :=FALSE;
	GVL_Main.M22.bHardwareEnable:= TRUE;
	GVL_Main.M22.bPowerSelf:= TRUE;
	GVL_Main.M22.nBrakeMode:= ENUM_StageBrakeMode.NO_BRAKE;
	GVL_Main.M23.bHardwareEnable:= TRUE;
	GVL_Main.M23.bPowerSelf:= TRUE;
	GVL_Main.M23.nBrakeMode:= ENUM_StageBrakeMode.NO_BRAKE;
	GVL_Main.M24.bHardwareEnable:= TRUE;
	GVL_Main.M24.bPowerSelf:= TRUE;
	GVL_Main.M24.nBrakeMode:= ENUM_StageBrakeMode.NO_BRAKE;
END_IF;


fbMotionXDC(stMotionStage:= GVL_Main.M22);
fbMotionRyDC(stMotionStage:= GVL_Main.M23);
fbMotionZDC(stMotionStage:= GVL_Main.M24);

END_PROGRAM

// ---- POUs/PRG_DET_SLIT.TcPOU
PROGRAM PRG_DET_SLIT
VAR
	fbSlits_Det: FB_Slits;
	bExecuteMotion: BOOL := FALSE;
	bMoveOk: BOOL;
END_VAR

// 4 jaws slit
fbSlits_Det(	i_DevName:=					'DET_SLITS',
				stTopBlade:=				GVL_Main.M20,
				stBottomBlade:=				GVL_Main.M21,
				stLeftBlade:=				GVL_Main.M18,
				stRightBlade:=				GVL_Main.M19,
				io_fbFFHWO:=				GVL_PMPS.io_fbFFHWO,
				fbArbiter:=					GVL_PMPS.fbArbiter,
				bExecuteMotion:=			bExecuteMotion,
				bMoveOk:=					bMoveOk
);

END_PROGRAM

// ---- POUs/FB_Slits.TcPOU
FUNCTION_BLOCK FB_Slits
VAR_IN_OUT
    stTopBlade: DUT_MotionStage;
    stBottomBlade: DUT_MotionStage;
    stLeftBlade: DUT_MotionStage; // Left Slit from upstream view
    stRightBlade: DUT_MotionStage; // Right Slit from upstream view
    bExecuteMotion:BOOL ;
    io_fbFFHWO    :    FB_HardwareFFOutput;
    fbArbiter: FB_Arbiter();
END_VAR

VAR_INPUT

    {attribute 'pytmc' := '
    pv: PMPS_OK;
    io: i;
    field: ZNAM False
    field: ONAM True
    '}
    bMoveOk:BOOL;

    (*Offsets*)
    {attribute 'pytmc' := '
    pv: Offset_Top;
    io: io;
    '}
    rEncoderOffsetTop: REAL;
    {attribute 'pytmc' := '
    pv: ZeroOffset_Bottom;
    io: io;
    '}
    rEncoderOffsetBottom: REAL;

    {attribute 'pytmc' := 'pv: ZeroOffset_Left; io: io;'}
    rEncoderOffsetLeft: REAL;
	
    {attribute 'pytmc' := '
    pv: ZeroOffset_Right;
    io: io;
    '}
    rEncoderOffsetRight: REAL;
    i_DevName : STRING; //device name for FFO and PMPS diagnostics
    {attribute 'pytmc' := '
    pv: Home;
    io: i;
    field: ZNAM False
    field: ONAM True
    '}
    bHome:BOOL:=FALSE;
END_VAR

VAR
    fbTopBlade: FB_MotionStage;
    fbBottomBlade: FB_MotionStage;
    fbLeftBlade: FB_MotionStage;
    fbRightBlade: FB_MotionStage;
    fPosTopBlade: LREAL;
    fPosBottomBlade: LREAL;
    fPosLeftBlade: LREAL;
    fPosRightBlade: LREAL;

	bCollisionLimitationVert: BOOL;
	bCollisionLimitationHorz: BOOL;
	
    (*Motion Parameters*)
    fSmallDelta: LREAL := 0.01;
    fBigDelta: LREAL := 20;
    fMaxVelocity: LREAL := 0.5;
    fHighAccel: LREAL := 0.8;
    fLowAccel: LREAL := 0.1;

    stTop: DUT_PositionState;
    stBOTTOM: DUT_PositionState;
    stLeft: DUT_PositionState;
    stRight: DUT_PositionState;

    {attribute 'pytmc' := 'pv: TOP'}
    fbTop: FB_StatePTPMove;
    {attribute 'pytmc' := 'pv: BOTTOM'}
    fbBottom: FB_StatePTPMove;
    {attribute 'pytmc' := 'pv: LEFT'}
    fbLeft: FB_StatePTPMove;
    {attribute 'pytmc' := 'pv: RIGHT'}
    fbRight: FB_StatePTPMove;

    (*EPICS pvs*)
    {attribute 'pytmc' := '
    pv: XWID_REQ;
    io: io;
    '}
    rReqApertureSizeX : REAL;
    {attribute 'pytmc' := '
    pv: YWID_REQ;
    io: io;
    '}
    rReqApertureSizeY : REAL;
    {attribute 'pytmc' := '
    pv: XCEN_REQ;
    io: io;
    '}
    rReqCenterX: REAL;
    {attribute 'pytmc' := '
    pv: YCEN_REQ;
    io: io;
    '}
    rReqCenterY: REAL;

    {attribute 'pytmc' := '
    pv: ACTUAL_XWIDTH;
    io: io;
    '}
    rActApertureSizeX : REAL;

    {attribute 'pytmc' := '
    pv: ACTUAL_YWIDTH;
    io: io;
    '}
    rActApertureSizeY : REAL;
    {attribute 'pytmc' := '
    pv: ACTUAL_XCENTER;
    io: io;
    '}
    rActCenterX: REAL;
    {attribute 'pytmc' := '
    pv: ACTUAL_YCENTER;
    io: io;
    '}
    rActCenterY: REAL;

    {attribute 'pytmc' := '
    pv: XCEN_SETZERO;
    io: io;
    '}
    rSetCenterX: BOOL;
    {attribute 'pytmc' := '
    pv: YCEN_SETZERO;
    io: io;
    '}
    rSetCenterY: BOOL;


    {attribute 'pytmc' := '
    pv: OPEN;
    io: io;
    field: ZNAM False
    field: ONAM True
    '}
    bOpen: BOOL;

    {attribute 'pytmc' := '
    pv: CLOSE;
    io: io;
    field: ZNAM False
    field: ONAM True
    '}
    bClose: BOOL;

    {attribute 'pytmc' := '
    pv: BLOCK;
    io: io;
    field: ZNAM False
    field: ONAM True
    '}
    bBlock: BOOL;


     {attribute 'pytmc' := '
    pv: HOME_READY;
    io: i;
    field: ZNAM False
    field: ONAM True
    '}
    bHomeReady:BOOL:=FALSE;


    //Local variables
    bInit: BOOL :=true;
    rTrig_Block: R_TRIG;
    rTrig_Open: R_TRIG;
    rTrig_Close: R_TRIG;

    //old values
    rOldReqApertureSizeX : REAL;
    rOldReqApertureSizeY : REAL;
    rOldReqCenterX: REAL;
    rOldReqCenterY: REAL;

    bExecuteMotionX: BOOL;
    bExecuteMotionY: BOOL;


    fPosBlock: LREAL;
    fPosClose: LREAL;
    fPosOpen: LREAL;

    stSetPositionOptions:ST_SetPositionOptions;
    fbSetPosition_TOP: MC_SetPosition;
    fbSetPosition_Bottom: MC_SetPosition;
    fbSetPosition_Left: MC_SetPosition;
    fbSetPosition_Right: MC_SetPosition;

    // For logging
    fbLogger : FB_LogMessage := (eSubsystem:=E_SubSystem.MOTION);
    tErrorPresent : R_TRIG;
    tAction : R_TRIG;
    tOverrideActivated : R_TRIG;

    FFO    :    FB_FastFault :=(
        i_DevName := 'Slits',
        i_Desc := 'Fault occurs when center is greated than that requested',
        i_TypeCode := 16#1010);


    bTest: BOOL;

    AptArrayStatus AT %Q* : ST_PMPS_Aperture_IO;
    AptArrayReq AT %I* : ST_PMPS_Aperture_IO;

	fbPower: MC_Power;
END_VAR

// Initialize
ACT_init();
// Instantiate Function block for all the blades
ACT_Motion();
//SET and GET the requested and Actual values
ACT_CalculatePositions();

// Software Limits to protect blades
ACT_VirtualLimitSW();

ACTION ACT_BLOCK:
rTrig_Block (CLK:= bBlock);
rTrig_Open (CLK:= bOpen);
rTrig_Close (CLK:= bClose);

if (rTrig_Block.Q) THEN
    //BLOCK

    bBlock := false;
END_IF

if (rTrig_Open.Q) THEN


    bOpen := false;
END_IF

if (rTrig_Close.Q) THEN


    bClose := false;
END_IF
END_ACTION

ACTION ACT_CalculatePositions:
//check if requested center or gap has changed
//check that the requested values are within acceptable motion range
IF (rOldReqApertureSizeX <> rReqApertureSizeX) THEN
        rOldReqApertureSizeX := rReqApertureSizeX;
        bExecuteMotionX := TRUE;
        fbLogger(sMsg:='Requested new X gap.', eSevr:=TcEventSeverity.Verbose);
END_IF

IF (rOldReqCenterX <> rReqCenterX) THEN
    rOldReqCenterX := rReqCenterX;
    bExecuteMotionX := TRUE;
    fbLogger(sMsg:='Requested new X center', eSevr:=TcEventSeverity.Verbose);
   // ELSE
      //  rReqCenterX := rActCenterX;
END_IF

IF (rOldReqApertureSizeY <> rReqApertureSizeY) THEN
        rOldReqApertureSizeY := rReqApertureSizeY;
        bExecuteMotionY := TRUE;
        fbLogger(sMsg:='Requested new Y gap.', eSevr:=TcEventSeverity.Verbose);

END_IF

IF (rOldReqCenterY <> rReqCenterY) THEN
    rOldReqCenterY := rReqCenterY;
    bExecuteMotionY := TRUE;
    fbLogger(sMsg:='Requested new Y center.', eSevr:=TcEventSeverity.Verbose);
   // ELSE
      //  rReqCenterY := rActCenterY;
END_IF


//Calculate requested target positions from requested gap and center
fPosTopBlade := (rReqApertureSizeY/2) + (rReqCenterY + rEncoderOffsetTop) ;
fPosBottomBlade := (-1*rReqApertureSizeY/2) + (rReqCenterY+rEncoderOffsetBottom);

fPosLeftBlade := (rReqApertureSizeX/2) + (rReqCenterX + rEncoderOffsetLeft);
fPosRightBlade := (-1*rReqApertureSizeX/2) + (rReqCenterX + rEncoderOffsetRight);


//Calculate actual gap and center from actual stages positions
rActApertureSizeX := LREAL_TO_REAL((stLeftBlade.stAxisStatus.fActPosition - rEncoderOffsetLeft) - (stRightBlade.stAxisStatus.fActPosition- rEncoderOffsetRight));

rActApertureSizeY := LREAL_TO_REAL((stTopBlade.stAxisStatus.fActPosition - rEncoderOffsetTop) - (stBottomBlade.stAxisStatus.fActPosition - rEncoderOffsetBottom));

rActCenterX := LREAL_TO_REAL((((stLeftBlade.stAxisStatus.fActPosition - rEncoderOffsetLeft)  + (stRightBlade.stAxisStatus.fActPosition - rEncoderOffsetRight ))/2));

rActCenterY := LREAL_TO_REAL((((stTopBlade.stAxisStatus.fActPosition - rEncoderOffsetTop) + (stBottomBlade.stAxisStatus.fActPosition - rEncoderOffsetBottom))/2));


// Prevent collision
bCollisionLimitationHorz	:= (rActApertureSizeX > -0.1);
bCollisionLimitationVert	:= (rActApertureSizeY > -0.1);
END_ACTION

ACTION ACT_Init:

//  init the motion stages parameters
IF ( bInit) THEN
    stTopBlade.bHardwareEnable := TRUE;
    stBottomBlade.bHardwareEnable := TRUE;
    stLeftBlade.bHardwareEnable := TRUE;
    stRightBlade.bHardwareEnable := TRUE;
    stTopBlade.bPowerSelf :=FALSE;
    stBottomBlade.bPowerSelf :=FALSE;
    stLeftBlade.bPowerSelf :=FALSE;
    stRightBlade.bPowerSelf :=FALSE;
    stTopBlade.nBrakeMode := ENUM_StageBrakeMode.NO_BRAKE;
    stBottomBlade.nBrakeMode := ENUM_StageBrakeMode.NO_BRAKE;
    stLeftBlade.nBrakeMode := ENUM_StageBrakeMode.NO_BRAKE;
    stRightBlade.nBrakeMode := ENUM_StageBrakeMode.NO_BRAKE;
    FFO.i_DevName := i_DevName;
END_IF
END_ACTION

ACTION ACT_Motion:
// Instantiate Function block for all the blades
fbTopBlade(stMotionStage:=stTopBlade);
fbBottomBlade(stMotionStage:=stBottomBlade);
fbLeftBlade(stMotionStage:=stLeftBlade);
fbRightBlade(stMotionStage:=stRightBlade);



// PTP Motion for each blade
stTop.sName := 'Top';
stTop.fPosition := fPosTopBlade;
stTop.fDelta := fSmallDelta;
stTop.fVelocity := fMaxVelocity;
stTop.fAccel := fHighAccel;
stTop.fDecel := fHighAccel;

stBOTTOM.sName := 'Bottom';
stBOTTOM.fPosition := fPosBottomBlade;
stBOTTOM.fDelta := fSmallDelta;
stBOTTOM.fVelocity := fMaxVelocity;
stBOTTOM.fAccel := fHighAccel;
stBOTTOM.fDecel := fHighAccel;

stLeft.sName := 'Left';
stLeft.fPosition := fPosLeftBlade;
stLeft.fDelta := fSmallDelta;
stLeft.fVelocity := fMaxVelocity;
stLeft.fAccel := fHighAccel;
stLeft.fDecel := fHighAccel;

stRight.sName := 'Right';
stRight.fPosition := fPosRightBlade;
stRight.fDelta := fSmallDelta;
stRight.fVelocity := fMaxVelocity;
stRight.fAccel := fHighAccel;
stRight.fDecel := fHighAccel;

IF (bExecuteMotionY) THEN
    fbTop.bExecute := fbBottom.bExecute := bExecuteMotionY;
    bExecuteMotionY:= FALSE;
END_IF

IF (bExecuteMotionX) THEN
    fbLeft.bExecute := fbRight.bExecute := bExecuteMotionX;
    bExecuteMotionX:= FALSE;
END_IF


fbTop(
    stPositionState:=stTop,
    bMoveOk:=bMoveOk,
    stMotionStage:=stTopBlade);

fbBottom(
    stPositionState:=stBOTTOM,
    bMoveOk:=bMoveOk,
    stMotionStage:=stBottomBlade);

fbLeft(
    stPositionState:=stLeft,
    bMoveOk:=bMoveOk,
    stMotionStage:=stLeftBlade);

fbRight(
    stPositionState:=stRight,
    bMoveOk:=bMoveOk,
    stMotionStage:=stRightBlade);
END_ACTION

ACTION ACT_VirtualLimitSW:

// Force set to false
stLeftBlade.bPowerSelf := stRightBlade.bPowerSelf := stTopBlade.bPowerSelf := stBottomBlade.bPowerSelf := FALSE;

// Set SafetyReady flags manually
stTopBlade.bSafetyReady:= TRUE;
stBottomBlade.bSafetyReady:= TRUE;
stLeftBlade.bSafetyReady:= TRUE;
stRightBlade.bSafetyReady:= TRUE;


// Note: FB_MotionStage calls FB_SetEnables internally that overwrites .bAllForwardEnable/.bAllBackwardEnable flags

fbPower(
	Axis := stTopBlade.Axis,
	Enable := stTopBlade.bAllEnable,
	Enable_Positive := stTopBlade.bAllForwardEnable,
	Enable_Negative := stTopBlade.bAllBackwardEnable AND bCollisionLimitationVert,
	Override := 100.000
);
fbPower(
	Axis := stBottomBlade.Axis,
	Enable := stBottomBlade.bAllEnable,
	Enable_Positive := stBottomBlade.bAllForwardEnable AND bCollisionLimitationVert,
	Enable_Negative := stBottomBlade.bAllBackwardEnable,
	Override := 100.000
);
fbPower(
	Axis := stLeftBlade.Axis,
	Enable := stLeftBlade.bAllEnable,
	Enable_Positive := stLeftBlade.bAllForwardEnable,
	Enable_Negative := stLeftBlade.bAllBackwardEnable AND bCollisionLimitationHorz,
	Override := 100.000
);
fbPower(
	Axis := stRightBlade.Axis,
	Enable := stRightBlade.bAllEnable,
	Enable_Positive := stRightBlade.bAllForwardEnable AND bCollisionLimitationHorz,
	Enable_Negative := stRightBlade.bAllBackwardEnable,
	Override := 100.000
);
END_ACTION

END_FUNCTION_BLOCK

// ---- POUs/PRG_DET_FRAME.TcPOU
PROGRAM PRG_DET_FRAME
VAR
	bInit: BOOL := TRUE;
	bError: BOOL := FALSE;
	bBusy: BOOL;
	bResetError: BOOL := FALSE;
	bEnableMotion : BOOL;
	bEnableMotion_M15 : BOOL;
	bEnableMotion_M16 : BOOL;
	bEnableMotion_M17 : BOOL;
	bEnableSetGaugeValue: BOOL;
	bEnableMoveRelative: BOOL;
	bEnableJackOff: BOOL;
	bEnableLevitation: BOOL;
	bEnableLanding: BOOL;
	bEnableAdjustingRoll: BOOL;
	bEnableAdjustingPitch: BOOL;
	bEnableAdjustingHeight: BOOL;
	
	bDone_M15, bDone_M16, bDone_M17: BOOL;
	
	tonWaitToStabilize: TON;

	tonSV2Open: TON;
	tonSV1Close: TON;
	
	tonDelayTrig: TON;
	
	iStepJackOff: INT := 1;
	iStepAdjustingRoll : INT := 1;
	iStepSetGaugeValue : INT := 1;
	iStepMoveRelative : INT := 1;
	iStepAdjustingPitch : INT := 1;
	iStepAdjustingHeight : INT := 1;
	
	trigDone: F_TRIG;
	
	fDistanceX: LREAL := 2.114; // in m
	fDistanceZ: LREAL := 2.142; // in m
	
	fbPower_AxisM15: MC_Power;
	fbPower_AxisM16: MC_Power;
	fbPower_AxisM17: MC_Power;
	
	fbSetPosition_M15: MC_SetPosition;
	fbSetPosition_M16: MC_SetPosition;
	fbSetPosition_M17: MC_SetPosition;

	fTargetPos_M15, fTargetPos_M16, fTargetPos_M17: LREAL;
	
    fbMoveRelative_M15: MC_MoveRelative;
    fbMoveRelative_M16: MC_MoveRelative;
    fbMoveRelative_M17: MC_MoveRelative;
END_VAR

// Read axis status
GVL_Main.M15.Axis.ReadStatus();
GVL_Main.M16.Axis.ReadStatus();
GVL_Main.M17.Axis.ReadStatus();

fbPower_AxisM15(
	Enable := GVL_Main.M15.bEnable,
	Enable_Positive := GVL_Main.M15.bLimitForwardEnable,
	Enable_Negative := GVL_Main.M15.bLimitBackwardEnable,
	Override := 100.000,
	Axis := GVL_Main.M15.Axis
);

fbPower_AxisM16(
	Enable := GVL_Main.M16.bEnable,
	Enable_Positive := GVL_Main.M16.bLimitForwardEnable,
	Enable_Negative := GVL_Main.M16.bLimitBackwardEnable,
	Override := 100.000,
	Axis := GVL_Main.M16.Axis
);

fbPower_AxisM17(
	Enable := GVL_Main.M17.bEnable,
	Enable_Positive := GVL_Main.M17.bLimitForwardEnable,
	Enable_Negative := GVL_Main.M17.bLimitBackwardEnable,
	Override := 100.000,
	Axis := GVL_Main.M17.Axis
);

GVL_Sensor.bFloating := GVL_Sensor.stPS1.fValue > 0.3 AND GVL_Sensor.stPS2.fValue > 0.18 AND GVL_Sensor.stPS3.fValue > 0.15;	

ACT_1_JACK_OFF();
ACT_2_Levitation();
ACT_3_Landing();
ACT_4_AdjustingRoll();
ACT_5_AdjustingPitch();
ACT_6_AdjustingHeight();
ACT_INIT();
ACT_SetGaugeValue();
ACT_MoveRelative();
ACT_ResetError();

ACTION ACT_1_JACK_OFF:
CASE iStepJackOff OF
	1:
		IF bEnableJackOff AND NOT(bBusy AND bError) THEN
			// Step1 read and apply gauge value
			bEnableSetGaugeValue := TRUE;
			iStepJackOff := 2;
		ELSE
			bEnableJackOff := FALSE;
		END_IF;
	2: 
		// Step2 wait until done
		IF NOT bEnableSetGaugeValue THEN
			// read latest status
			GVL_Main.M15.Axis.ReadStatus();
			GVL_Main.M16.Axis.ReadStatus();
			GVL_Main.M17.Axis.ReadStatus();
			IF abs(GVL_Main.M15.Axis.NcToPlc.ActPos) < 0.1 AND abs(GVL_Main.M16.Axis.NcToPlc.ActPos) < 0.1 AND abs(GVL_Main.M17.Axis.NcToPlc.ActPos) < 0.1 THEN
				// We dont need to move any more....
				iStepJackOFF := 5;
			ELSIF max(GVL_Main.M15.Axis.NcToPlc.ActPos, GVL_Main.M16.Axis.NcToPlc.ActPos, GVL_Main.M17.Axis.NcToPlc.ActPos)
				- min(GVL_Main.M15.Axis.NcToPlc.ActPos, GVL_Main.M16.Axis.NcToPlc.ActPos, GVL_Main.M17.Axis.NcToPlc.ActPos) > 10.0 THEN
				// Some axis may be step-out...
				iStepJackOFF := -1;
			ELSE
				iStepJackOff := 3;
			END_IF;
		END_IF;
	3: 
		// Step3 calcurate motion distance		
		fTargetPos_M15 := -1 * GVL_Main.M15.Axis.NcToPlc.ActPos;
		fTargetPos_M16 := -1 * GVL_Main.M16.Axis.NcToPlc.ActPos;
		fTargetPos_M17 := -1 * GVL_Main.M17.Axis.NcToPlc.ActPos;
		
		// Enable Relative Motion Act
		bEnableMoveRelative := TRUE;
		
		iStepJackOff := 4;
	4: 
		// Wait until Done.
		IF NOT bEnableMoveRelative THEN
			// read and apply gauge value
			bEnableSetGaugeValue := TRUE;
			iStepJackOff := 2;
		END_IF;
	5:
		// End
		bEnableJackOff:= FALSE;
		bBusy := FALSE;
		iStepJackOff:=1;
	-1:
		// Error
		bError:= TRUE;
		bEnableJackOff:= FALSE;
		bBusy := FALSE;
		iStepJackOff:=1;
END_CASE;
END_ACTION

ACTION ACT_2_Levitation:

IF bEnableLevitation THEN
	IF GVL_Sensor.stPS1.fValue > 0.15 AND GVL_Sensor.stPS2.fValue > 0.15 THEN
		GVL_Main.bOpenSV1 := TRUE;
	END_IF;
END_IF;


// SV2 will open after 3 secounds from SV1 opened...
tonSV2Open(
	IN := bEnableLevitation AND GVL_Main.bOpenSV1,
	PT := T#3s
);

IF tonSV2Open.Q THEN
	GVL_Main.bOpenSV2 := TRUE;
	bEnableLevitation := FALSE;
END_IF;
END_ACTION

ACTION ACT_3_Landing:


IF bEnableLanding AND NOT (bBusy OR bError) THEN
	GVL_Main.bOpenSV2 := FALSE;
	bBusy:= TRUE;
END_IF;

tonSV1Close(
	IN := bEnableLanding AND NOT GVL_Main.bOpenSV2,
	PT := T#3s
);

IF tonSV1Close.Q THEN
	GVL_Main.bOpenSV1 := FALSE;
	bEnableLanding := FALSE;
	bBusy:= FALSE;
END_IF;
END_ACTION

ACTION ACT_4_AdjustingRoll:
CASE iStepAdjustingRoll OF
	1:
		IF bEnableAdjustingRoll AND NOT(bBusy AND bError) THEN
			// Step1 read and apply gauge value
			bEnableSetGaugeValue := TRUE;
			iStepAdjustingRoll := 2;
		ELSE
			bEnableAdjustingRoll := FALSE;
		END_IF;
	2: 
		// Step2 wait until done
		IF NOT bEnableSetGaugeValue THEN
			iStepAdjustingRoll := 3;
		END_IF;
	3: 
		// Step3 calcurate motion distance
		// read latest status
		GVL_Main.M15.Axis.ReadStatus();
		GVL_Main.M16.Axis.ReadStatus();
		GVL_Main.M17.Axis.ReadStatus();
				
		IF GVL_Sensor.stFrameR.fValue > 0 THEN
			// Need to up YDF1
			fTargetPos_M15 := abs(REAL_TO_LREAL(GVL_Sensor.stFrameR.fValue)) * fDistanceX / 2 * 0.9;
			fTargetPos_M16 := 0;
			fTargetPos_M17 := 0;
			// Enable Relative Motion Act
			bEnableMoveRelative := TRUE;
			iStepAdjustingRoll := 4;
		ELSE
			// Need to up YDF2
			fTargetPos_M15 := 0;
			fTargetPos_M16 := abs(REAL_TO_LREAL(GVL_Sensor.stFrameR.fValue)) * fDistanceX / 2 * 0.9;
			fTargetPos_M17 := 0;
			// Enable Relative Motion Act
			bEnableMoveRelative := TRUE;
			iStepAdjustingRoll := 4;
		END_IF;
	4: 
		// Wait until Done. and wait tilt sensor stabilization.
		tonWaitToStabilize(IN:=NOT bEnableMoveRelative, PT:=T#5s);
		IF tonWaitToStabilize.Q THEN
			iStepAdjustingRoll := 5;
			tonWaitToStabilize(IN:=FALSE);
		END_IF;
	5:
		IF abs(GVL_Sensor.stFrameR.fValue) > 0.05 THEN
			// Iterartion
			bEnableSetGaugeValue := TRUE;
			iStepAdjustingRoll := 2;
		ELSE
			// End
			bEnableAdjustingRoll:= FALSE;
			iStepAdjustingRoll:=1;
		END_IF;
	-1:
		// Error
		bError:= TRUE;
		bEnableAdjustingRoll:= FALSE;
		iStepAdjustingRoll:=1;
END_CASE;
END_ACTION

ACTION ACT_5_AdjustingPitch:
CASE iStepAdjustingPitch OF
	1:
		IF bEnableAdjustingPitch AND NOT(bBusy AND bError) THEN
			// Step1 read and apply gauge value
			bEnableSetGaugeValue := TRUE;
			iStepAdjustingPitch := 2;
		ELSE
			bEnableAdjustingPitch := FALSE;
		END_IF;
	2: 
		// Step2 wait until done
		IF NOT bEnableSetGaugeValue THEN
			iStepAdjustingPitch := 3;
		END_IF;
	3: 
		// Step3 calcurate motion distance
		// read latest status
		GVL_Main.M15.Axis.ReadStatus();
		GVL_Main.M16.Axis.ReadStatus();
		GVL_Main.M17.Axis.ReadStatus();
				
		IF GVL_Sensor.stFrameP.fValue > 0 THEN
			// Need to up YDF1 AND 2
			fTargetPos_M15 := abs(REAL_TO_LREAL(GVL_Sensor.stFrameP.fValue)) * fDistanceZ / 2 * 0.9;
			fTargetPos_M16 := abs(REAL_TO_LREAL(GVL_Sensor.stFrameP.fValue)) * fDistanceZ / 2 * 0.9;;
			fTargetPos_M17 := 0;
			// Enable Relative Motion Act
			bEnableMoveRelative := TRUE;
			iStepAdjustingPitch := 4;
		ELSE
			// Need to up YDF3
			fTargetPos_M15 := 0;
			fTargetPos_M16 := 0;
			fTargetPos_M17 := abs(REAL_TO_LREAL(GVL_Sensor.stFrameP.fValue)) * fDistanceZ / 2 * 0.9;
			// Enable Relative Motion Act
			bEnableMoveRelative := TRUE;
			iStepAdjustingPitch := 4;
		END_IF;
	4: 
		// Wait until Done. and wait tilt sensor stabilization.
		tonWaitToStabilize(IN:=NOT bEnableMoveRelative, PT:=T#5s);
		IF tonWaitToStabilize.Q THEN
			iStepAdjustingPitch := 5;
		END_IF;
	5:
		IF abs(GVL_Sensor.stFrameP.fValue) > 0.05 THEN
			// Iteration
			bEnableSetGaugeValue := TRUE;
			iStepAdjustingPitch := 2;
		ELSE
			// End
			bEnableAdjustingPitch:= FALSE;
			iStepAdjustingPitch:=1;
		END_IF;
	-1:
		// Error
		bError:= TRUE;
		bEnableAdjustingPitch:= FALSE;
		iStepAdjustingPitch:=1;
END_CASE;
END_ACTION

ACTION ACT_6_AdjustingHeight:
CASE iStepAdjustingHeight OF
	1:
		IF bEnableAdjustingHeight AND NOT(bBusy AND bError) THEN
			// Step1 read and apply gauge value
			bEnableSetGaugeValue := TRUE;
			iStepAdjustingHeight := 2;
		ELSE
			bEnableAdjustingHeight := FALSE;
		END_IF;
	2: 
		// Step2 wait until done
		IF NOT bEnableSetGaugeValue THEN
			iStepAdjustingHeight := 3;
		END_IF;
	3: 
		// Step3 calcurate motion distance
		// read latest status
		GVL_Main.M15.Axis.ReadStatus();
		GVL_Main.M16.Axis.ReadStatus();
		GVL_Main.M17.Axis.ReadStatus();

		// Need to move YDF 1~3
		fTargetPos_M15 := -1 * REAL_TO_LREAL(GVL_Sensor.stHDF.fValue) * 0.9;
		fTargetPos_M16 := -1 * REAL_TO_LREAL(GVL_Sensor.stHDF.fValue) * 0.9;
		fTargetPos_M17 := -1 * REAL_TO_LREAL(GVL_Sensor.stHDF.fValue) * 0.9;
		// Enable Relative Motion Act
		bEnableMoveRelative := TRUE;
		iStepAdjustingHeight := 4;

	4: 
		// Wait until Done. and wait tilt sensor stabilization.
		tonWaitToStabilize(IN:=NOT bEnableMoveRelative, PT:=T#5s);
		IF tonWaitToStabilize.Q THEN
			iStepAdjustingHeight := 5;
		END_IF;
	5:
		// check pitch and roll (if some axis is step-out)
		IF abs(GVL_Sensor.stFrameP.fValue) > 0.5 OR abs(GVL_Sensor.stFrameR.fValue) > 0.5 THEN
			bError := TRUE;
		END_IF;		
		
		IF abs(GVL_Sensor.stHDF.fValue) > 0.05 AND NOT bError THEN
			// Iteration
			bEnableAdjustingHeight := FALSE;
			iStepAdjustingHeight := 2;
		ELSE
			// End
			bEnableAdjustingHeight:= FALSE;
			iStepAdjustingHeight:=1;
		END_IF;
	-1:
		// Error
		bError:= TRUE;
		bEnableAdjustingHeight:= FALSE;
		iStepAdjustingHeight:=1;
END_CASE;
END_ACTION

ACTION ACT_INIT:
IF bINIT THEN
	bINIT := FALSE;
	
	GVL_Main.M15.nBrakeMode := ENUM_StageBrakeMode.NO_BRAKE;
	GVL_Main.M15.bHardwareEnable := TRUE;
	GVL_Main.M15.bPowerSelf := TRUE;
	GVL_Main.M16.nBrakeMode := ENUM_StageBrakeMode.NO_BRAKE;
	GVL_Main.M16.bHardwareEnable := TRUE;
	GVL_Main.M16.bPowerSelf := TRUE;
	GVL_Main.M17.nBrakeMode := ENUM_StageBrakeMode.NO_BRAKE;
	GVL_Main.M17.bHardwareEnable := TRUE;
	GVL_Main.M17.bPowerSelf := TRUE;
	
	// Read linear gauge value
	bEnableSetGaugeValue := TRUE;

END_IF;
END_ACTION

ACTION ACT_MoveRelative:
CASE iStepMoveRelative OF
	1: 
		IF bEnableMoveRelative AND NOT (bBusy OR bError) THEN
			bBusy:= TRUE;
			bEnableMotion := TRUE;
			bDone_M15 := bDone_M16 := bDone_M17 := FALSE;
			iStepMoveRelative:= 2;
		ELSE
			bEnableMoveRelative:= FALSE;
		END_IF;
	2:
		// Step2 Execute motion
		IF fbMoveRelative_M15.Error OR fbMoveRelative_M16.Error OR fbMoveRelative_M17.Error THEN
			iStepMoveRelative:= -1;
			bError := 1;
		END_IF;
		
		IF (bDone_M15 AND bDone_M16 AND bDone_M17) AND NOT(fbMoveRelative_M15.Execute OR fbMoveRelative_M16.Execute OR fbMoveRelative_M17.Execute) THEN
			iStepMoveRelative:= 3;
		END_IF;
		
		IF fbMoveRelative_M15.Done THEN
			bDone_M15 := TRUE;
		END_IF;
		IF fbMoveRelative_M16.Done THEN
			bDone_M16 := TRUE;
		END_IF;
		IF fbMoveRelative_M17.Done THEN
			bDone_M17 := TRUE;
		END_IF;
		
		fbMoveRelative_M15(	Axis		:= GVL_Main.M15.Axis,
							Execute		:= bEnableMotion AND NOT (bDone_M15 OR bError),
							Distance	:= fTargetPos_M15,
							Velocity	:= 0.05,
							Acceleration:= 0.8,
							Deceleration:= 0.8,
							Jerk		:= 32
		);
		fbMoveRelative_M16(	Axis		:= GVL_Main.M16.Axis,
							Execute		:= bEnableMotion AND NOT (bDone_M16 OR bError),
							Distance	:= fTargetPos_M16,
							Velocity	:= 0.05,
							Acceleration:= 0.8,
							Deceleration:= 0.8,
							Jerk		:= 32
		);
		fbMoveRelative_M17(	Axis		:= GVL_Main.M17.Axis,
							Execute		:= bEnableMotion AND NOT (bDone_M17 OR bError),
							Distance	:= fTargetPos_M17,
							Velocity	:= 0.05,
							Acceleration:= 0.8,
							Deceleration:= 0.8,
							Jerk		:= 32
		);
	3:
		// End
		bEnableMotion:= FALSE;
		bEnableMoveRelative:= FALSE;
		bBusy := FALSE;
		iStepMoveRelative:=1;
	-1:
		// Error
		fbMoveRelative_M15.Execute:= FALSE;
		fbMoveRelative_M16.Execute:= FALSE;
		fbMoveRelative_M17.Execute:= FALSE;
		bError:= TRUE;
		bEnableMotion:= FALSE;
		bEnableMoveRelative:= FALSE;
		bBusy := FALSE;
		iStepMoveRelative:=1;
END_CASE;
END_ACTION

ACTION ACT_ResetError:

IF bResetError THEN
	bResetError := FALSE;
	bError:= FALSE;
	bBusy:=FALSE;
	bEnableMotion := FALSE;
	bEnableMotion_M15 := FALSE;
	bEnableMotion_M16 := FALSE;
	bEnableMotion_M17 := FALSE;
	bEnableSetGaugeValue := FALSE;
	bEnableMoveRelative := FALSE;
	bEnableJackOff := FALSE;
	bEnableLevitation := FALSE;
	bEnableLanding := FALSE;
	bEnableAdjustingRoll := FALSE;
	bEnableAdjustingPitch := FALSE;
	bEnableAdjustingHeight := FALSE;
	
	bDone_M15 := bDone_M16 := bDone_M17 := FALSE;
	
	iStepJackOff := 1;
	iStepAdjustingRoll := 1;
	iStepSetGaugeValue := 1;
	iStepMoveRelative := 1;
	iStepAdjustingPitch := 1;
	iStepAdjustingHeight := 1;
END_IF;
END_ACTION

ACTION ACT_SetGaugeValue:

CASE iStepSetGaugeValue OF
	1:
		IF bEnableSetGaugeValue AND NOT (bBusy OR bError) THEN
			fTargetPos_M15 := GVL_Sensor.stYDF1.fValue;
			fTargetPos_M16 := GVL_Sensor.stYDF2.fValue;
			fTargetPos_M17 := GVL_Sensor.stYDF3.fValue;
			
			iStepSetGaugeValue:=2;
		ELSE
			bEnableSetGaugeValue := FALSE;
		END_IF;		
	2:		
		fbSetPosition_M15(	Axis :=		GVL_Main.M15.Axis,
							Execute :=	NOT fbSetPosition_M15.Done,
							Position :=	fTargetPos_M15
		);
		
		fbSetPosition_M16(	Axis :=		GVL_Main.M16.Axis,
							Execute :=	NOT fbSetPosition_M16.Done,
							Position :=	fTargetPos_M16
		);
		
		fbSetPosition_M17(	Axis :=		GVL_Main.M17.Axis,
							Execute :=	NOT fbSetPosition_M17.Done,
							Position :=	fTargetPos_M17
		);
		IF fbSetPosition_M15.Done OR fbSetPosition_M15.Error THEN
			fbSetPosition_M15(	Axis :=		GVL_Main.M15.Axis,
								Execute :=	FALSE
			);
		END_IF;
		IF fbSetPosition_M16.Done OR fbSetPosition_M16.Error THEN	
			fbSetPosition_M16(	Axis :=		GVL_Main.M16.Axis,
								Execute :=	FALSE
			);
		END_IF;
		IF fbSetPosition_M17.Done OR fbSetPosition_M17.Error THEN
			fbSetPosition_M17(	Axis :=		GVL_Main.M17.Axis,
								Execute :=	FALSE
			);
		END_IF;
		
		IF NOT(fbSetPosition_M17.Execute OR fbSetPosition_M17.Execute OR fbSetPosition_M17.Execute) THEN
			iStepSetGaugeValue:=3;
		END_IF;
		
	3:		
		bEnableSetGaugeValue := FALSE;
		iStepSetGaugeValue:=1;
END_CASE;
END_ACTION

END_PROGRAM

// ---- POUs/PRG_OPT_SLITS.TcPOU
PROGRAM PRG_OPT_SLITS
VAR
	fbSlits_Opt: FB_Slits;
	bExecuteMotion: BOOL := FALSE;
	bMoveOk: BOOL;
END_VAR

fbSlits_Opt(	i_DevName:=					'OPT_SLITS',
				stTopBlade:=				GVL_Main.M5,
				stBottomBlade:=				GVL_Main.M6,
				stLeftBlade:=				GVL_Main.M3,
				stRightBlade:=				GVL_Main.M4,
				io_fbFFHWO:=				GVL_PMPS.io_fbFFHWO,
				fbArbiter:=					GVL_PMPS.fbArbiter,
				bExecuteMotion:=			bExecuteMotion,
				bMoveOk:=					bMoveOk
);

END_PROGRAM

// ---- POUs/PRG_OPT_YG.TcPOU
PROGRAM PRG_OPT_YG
VAR
	bDebug: BOOL;
	bExecuteMotion: BOOL;
	bMoveOk: BOOL;
	fbYGMotion: FB_3AxesJack;
END_VAR

fbYGMotion(
	bExecuteMotion	:= bExecuteMotion,
	bMoveOk			:= bMoveOk,
	stJack1Axis		:= GVL_Main.M7,
	stJack2Axis		:= GVL_Main.M8,
	stJack3Axis		:= GVL_Main.M9,
	i_DevName		:= 'OPT_YG',
	io_fbFFHWO		:= GVL_PMPS.io_fbFFHWO,
	fbArbiter		:= GVL_PMPS.fbArbiter,
);

END_PROGRAM

// ---- POUs/FB_3AxesJack.TcPOU
FUNCTION_BLOCK FB_3AxesJack
VAR_IN_OUT
    stJack1Axis: DUT_MotionStage;
    stJack2Axis: DUT_MotionStage;
    stJack3Axis: DUT_MotionStage;
    bExecuteMotion:BOOL ;
    io_fbFFHWO    :    FB_HardwareFFOutput;
    fbArbiter: FB_Arbiter();
END_VAR
VAR_INPUT
	
    {attribute 'pytmc' := '
    pv: PMPS_OK;
    io: i;
    field: ZNAM False
    field: ONAM True
    '}
    bMoveOk:BOOL;

    (*Offsets*)
    {attribute 'pytmc' := '
    pv: ZeroOffset_Jack1;
    io: io;
    '}
    rEncoderOffsetJack1: REAL;
	
    {attribute 'pytmc' := '
    pv: ZeroOffset_Jack2;
    io: io;
    '}
    rEncoderOffsetJack2: REAL;
	
    {attribute 'pytmc' := '
    pv: ZeroOffset_Jack3;
    io: io;
    '}
    rEncoderOffsetJack3: REAL;
	
	(*Distance X*)
	rDistanceX: REAL := 0.24;
	(*Distance Z*)
	rDistanceZ: REAL := 0.88;
	
	(* Limit to Y +/-5mm and +/- Pitch/Roll 18mrad *)
	rLimitPositionMax: REAL := 5;
	rLimitPositionMin: REAL := -5;	
	rLimitPitchMin: REAL := -18;
	rLimitPitchMax: REAL :=  18;
	rLimitRollMin: REAL  := -18;
	rLimitRollMax: REAL  :=  18;

    i_DevName : STRING; //device name for FFO and PMPS diagnostics
	
     {attribute 'pytmc' := '
    pv: Home;
    io: i;
    field: ZNAM False
    field: ONAM True
    '}
    bHome:BOOL:=FALSE;
END_VAR

VAR
	fbJack1Stage: FB_MotionStage;
    fbJack2Stage: FB_MotionStage;
    fbJack3Stage: FB_MotionStage;
    fPosJack1Stage: LREAL;
    fPosJack2Stage: LREAL;
    fPosJack3Stage: LREAL;

    (*Motion Parameters*)
    fSmallDelta: LREAL := 0.01;
    fBigDelta: LREAL := 10;
    fMaxVelocity: LREAL := 0.05;
    fHighAccel: LREAL := 0.8;
    fLowAccel: LREAL := 0.1;

    stJack1: DUT_PositionState;
    stJack2: DUT_PositionState;
    stJack3: DUT_PositionState;

    {attribute 'pytmc' := 'pv: JACK1'}
    fbJack1: FB_StatePTPMove;
    {attribute 'pytmc' := 'pv: JACK2'}
    fbJack2: FB_StatePTPMove;
    {attribute 'pytmc' := 'pv: JACK3'}
    fbJack3: FB_StatePTPMove;

    (*EPICS pvs*)
    {attribute 'pytmc' := '
    pv: POS_REQ;
    io: io;
    '}
    rReqPosition : REAL;
	
    {attribute 'pytmc' := '
    pv: PIT_REQ;
    io: io;
    '}
    rReqPitch : REAL;
	
    {attribute 'pytmc' := '
    pv: ROL_REQ;
    io: io;
    '}
    rReqRoll : REAL;


    {attribute 'pytmc' := '
    pv: ACTUAL_POSISION;
    io: io;
    '}
    rActPosition : REAL;

    {attribute 'pytmc' := '
    pv: ACTUAL_PITCH;
    io: io;
    '}
    rActPitch : REAL;

    {attribute 'pytmc' := '
    pv: ACTUAL_ROLL;
    io: io;
    '}
    rActRoll : REAL;
	

    {attribute 'pytmc' := '
    pv: HOME_READY;
    io: i;
    field: ZNAM False
    field: ONAM True
    '}
    bHomeReady:BOOL:=FALSE;


    //Local variables
    bInit: BOOL :=true;

    //old values
    rOldReqPosition : REAL;
    rOldReqPitch: REAL;
    rOldReqRoll: REAL;

    bExecuteMotionX: BOOL;

	rPosAvgJAck1_3: REAL;

    fPosBlock: LREAL;
    fPosClose: LREAL;
    fPosOpen: LREAL;

    stSetPositionOptions: ST_SetPositionOptions;
    fbSetPosition_Pos: MC_SetPosition;
    fbSetPosition_Angle: MC_SetPosition;

    // For logging
    fbLogger : FB_LogMessage := (eSubsystem:=E_SubSystem.MOTION);
    tErrorPresent : R_TRIG;
    tAction : R_TRIG;
    tOverrideActivated : R_TRIG;

    FFO    :    FB_FastFault :=(
        i_DevName := '3Jack',
        i_Desc := 'Fault occurs when center is greated than that requested',
        i_TypeCode := 16#1010);


    bTest: BOOL;

    AptArrayStatus AT %Q* : ST_PMPS_Aperture_IO;
    AptArrayReq AT %I* : ST_PMPS_Aperture_IO;
	
	
	fbPower: MC_POWER;
END_VAR

// Initialize
ACT_init();

// Instantiate Function block for all the blades
ACT_Motion();

//SET and GET the requested and Actual values
ACT_CalculatePositions();

// Software Limits to protect blades
ACT_VirtualLimitSW();

ACTION ACT_CalculatePositions:
//check if requested center or gap has changed
//check that the requested values are within acceptable motion range
IF (rOldReqPosition <> rReqPosition) THEN
        rOldReqPosition := rReqPosition;
        bExecuteMotionX := TRUE;
        fbLogger(sMsg:='Requested new Position.', eSevr:=TcEventSeverity.Verbose);
END_IF

IF (rOldReqPitch <> rReqPitch) THEN
    rOldReqPitch := rReqPitch;
    bExecuteMotionX := TRUE;
    fbLogger(sMsg:='Requested new Pitch', eSevr:=TcEventSeverity.Verbose);
END_IF

IF (rOldReqRoll <> rReqRoll) THEN
    rOldReqRoll := rReqRoll;
    bExecuteMotionX := TRUE;
    fbLogger(sMsg:='Requested new Roll', eSevr:=TcEventSeverity.Verbose);
END_IF

//Calculate requested target positions from requested gap and center
fPosJack1Stage	:= rReqPosition + rDistanceX / 2 * rReqRoll + rDistanceZ / 2 * rReqPitch + rEncoderOffsetJack1;
fPosJack2Stage	:= rReqPosition - rDistanceX / 2 * rReqRoll + rEncoderOffsetJack2;
fPosJack3Stage	:= rReqPosition + rDistanceX / 2 * rReqRoll - rDistanceZ / 2 * rReqPitch + rEncoderOffsetJack3;

//Calculate actual gap and center from actual stages positions
rPosAvgJack1_3	:= LREAL_TO_REAL( ((stJack1Axis.stAxisStatus.fActPosition - rEncoderOffsetJack1) + (stJack3Axis.stAxisStatus.fActPosition - rEncoderOffsetJack3)) / 2 );
rActPosition	:= LREAL_TO_REAL( ((rPosAvgJAck1_3 + (stJack2Axis.stAxisStatus.fActPosition - rEncoderOffsetJack2)) / 2 ));
rActPitch		:= LREAL_TO_REAL( ((stJack1Axis.stAxisStatus.fActPosition - rEncoderOffsetJack1) - (stJack3Axis.stAxisStatus.fActPosition - rEncoderOffsetJack3)) / rDistanceZ);
rActRoll		:= LREAL_TO_REAL( (rActPosition - (stJack2Axis.stAxisStatus.fActPosition - rEncoderOffsetJack2)) / (rDistanceX/2)); // mrad
END_ACTION

ACTION ACT_Init:

//  init the motion stages parameters
IF ( bInit) THEN
    stJack1Axis.bHardwareEnable := TRUE;
    stJack2Axis.bHardwareEnable := TRUE;
    stJack3Axis.bHardwareEnable := TRUE;
    stJack1Axis.bPowerSelf :=FALSE;
    stJack2Axis.bPowerSelf :=FALSE;
    stJack3Axis.bPowerSelf :=FALSE;
    stJack1Axis.nBrakeMode := ENUM_StageBrakeMode.NO_BRAKE;
    stJack2Axis.nBrakeMode := ENUM_StageBrakeMode.NO_BRAKE;
    stJack3Axis.nBrakeMode := ENUM_StageBrakeMode.NO_BRAKE;
    FFO.i_DevName := i_DevName;
END_IF
END_ACTION

ACTION ACT_Motion:
// Instantiate Function block for all the blades
fbJack1Stage(stMotionStage:=stJack1Axis);
fbJack2Stage(stMotionStage:=stJack2Axis);
fbJack3Stage(stMotionStage:=stJack3Axis);



// PTP Motion for each blade
stJack1.sName := 'Jack1';
stJack1.fPosition := fPosJack1Stage;
stJack1.fDelta := fSmallDelta;
stJack1.fVelocity := fMaxVelocity;
stJack1.fAccel := fHighAccel;
stJack1.fDecel := fHighAccel;

stJack2.sName := 'Jack2';
stJack2.fPosition := fPosJack2Stage;
stJack2.fDelta := fSmallDelta;
stJack2.fVelocity := fMaxVelocity;
stJack2.fAccel := fHighAccel;
stJack2.fDecel := fHighAccel;

stJack3.sName := 'Jack3';
stJack3.fPosition := fPosJack3Stage;
stJack3.fDelta := fSmallDelta;
stJack3.fVelocity := fMaxVelocity;
stJack3.fAccel := fHighAccel;
stJack3.fDecel := fHighAccel;


IF (bExecuteMotionX) THEN
    fbJack1.bExecute := fbJack2.bExecute := fbJack3.bExecute := bExecuteMotionX;
    bExecuteMotionX:= FALSE;
END_IF


fbJack1(
    stPositionState:=stJack1,
    bMoveOk:=bMoveOk,
    stMotionStage:=stJack1Axis);

fbJack2(
    stPositionState:=stJack2,
    bMoveOk:=bMoveOk,
    stMotionStage:=stJack2Axis);
	
fbJack3(
    stPositionState:=stJack3,
    bMoveOk:=bMoveOk,
    stMotionStage:=stJack3Axis);
END_ACTION

ACTION ACT_VirtualLimitSW:

// Force set to false
stJack1Axis.bPowerSelf := stJack2Axis.bPowerSelf := stJack3Axis.bPowerSelf := FALSE;

// Set SafetyReady flags manually
stJack1Axis.bSafetyReady:= TRUE;
stJack2Axis.bSafetyReady:= TRUE;
stJack3Axis.bSafetyReady:= TRUE;


// Note: FB_MotionStage calls FB_SetEnables internally that overwrites .bAllForwardEnable/.bAllBackwardEnable flags

fbPower(
	Axis := stJack1Axis.Axis,
	Enable := stJack1Axis.bAllEnable,
	Enable_Positive := stJack1Axis.bAllForwardEnable  AND rActPosition <= rLimitPositionMax AND rActPitch <= rLimitPitchMax,
	Enable_Negative := stJack1Axis.bAllBackwardEnable AND rActPosition >= rLimitPositionMin AND rActPitch >= rLimitPitchMin,
	Override := 100.000
);
fbPower(
	Axis := stJack2Axis.Axis,
	Enable := stJack2Axis.bAllEnable,
	Enable_Positive := stJack2Axis.bAllForwardEnable  AND rActPosition <= rLimitPositionMax AND rActRoll >= rLimitRollMin,
	Enable_Negative := stJack2Axis.bAllBackwardEnable AND rActPosition >= rLimitPositionMin AND rActRoll <= rLimitRollMax,
	Override := 100.000
);
fbPower(
	Axis := stJack3Axis.Axis,
	Enable := stJack3Axis.bAllEnable,
	Enable_Positive := stJack3Axis.bAllForwardEnable  AND rActPosition <= rLimitPositionMax AND rActPitch >= rLimitPitchMin,
	Enable_Negative := stJack3Axis.bAllBackwardEnable AND rActPosition >= rLimitPositionMin AND rActPitch <= rLimitPitchMax,
	Override := 100.000
);
END_ACTION

END_FUNCTION_BLOCK

// ---- POUs/PRG_OPT_XPM.TcPOU
PROGRAM PRG_OPT_XPM
VAR
	bInit: BOOL;
	
	fb2AxesXPM: FB_2AxesTrans;
	bExecuteMotionXPM: BOOL;
	bMoveOkXPM: BOOL;
END_VAR


fb2AxesXPM(	i_DevName		:=	'OPT_XPM',
			stFirstAxis		:=	GVL_Main.M12,
			stSecondAxis	:=	GVL_Main.M13,
			bExecuteMotion	:=	bExecuteMotionXPM,
			io_fbFFHWO		:=	GVL_PMPS.io_fbFFHWO,
			fbArbiter		:=	GVL_PMPS.fbArbiter,
			rDistance		:=	0.4, // 0.4m
			bMoveOk			:= bMoveOkXPM
);

END_PROGRAM

// ---- POUs/FB_2AxesTrans.TcPOU
FUNCTION_BLOCK FB_2AxesTrans
VAR_IN_OUT
    stFirstAxis: DUT_MotionStage;
    stSecondAxis: DUT_MotionStage;
    bExecuteMotion:BOOL ;
    io_fbFFHWO    :    FB_HardwareFFOutput;
    fbArbiter: FB_Arbiter();
END_VAR
VAR_INPUT
	
    {attribute 'pytmc' := '
    pv: PMPS_OK;
    io: i;
    field: ZNAM False
    field: ONAM True
    '}
    bMoveOk:BOOL;

    (*Offsets*)
    {attribute 'pytmc' := '
    pv: ZeroOffset_First;
    io: io;
    '}
    rEncoderOffsetFirst: REAL;
	
    {attribute 'pytmc' := '
    pv: ZeroOffset_Secound;
    io: io;
    '}
    rEncoderOffsetSecound: REAL;
	
	(*Distance between 1st stage and 2nd stage*)
	rDistance: REAL := 0.40;

    i_DevName : STRING; //device name for FFO and PMPS diagnostics
	
     {attribute 'pytmc' := '
    pv: Home;
    io: i;
    field: ZNAM False
    field: ONAM True
    '}
    bHome:BOOL:=FALSE;
END_VAR
VAR
	fbFirstStage: FB_MotionStage;
    fbSecondStage: FB_MotionStage;
    fPosFirstStage: LREAL;
    fPosSecondStage: LREAL;

    (*Motion Parameters*)
    fSmallDelta: LREAL := 0.01;
    fBigDelta: LREAL := 10;
    fMaxVelocity: LREAL := 0.03;
    fHighAccel: LREAL := 0.8;
    fLowAccel: LREAL := 0.1;

    stFirst: DUT_PositionState;
    stSecond: DUT_PositionState;

    {attribute 'pytmc' := 'pv: FIRST'}
    fbFirst: FB_StatePTPMove;
    {attribute 'pytmc' := 'pv: SECOND'}
    fbSecond: FB_StatePTPMove;

    (*EPICS pvs*)
    {attribute 'pytmc' := '
    pv: POS_REQ;
    io: io;
    '}
    rReqPosition : REAL;
    {attribute 'pytmc' := '
    pv: ANG_REQ;
    io: io;
    '}
    rReqAngle : REAL;


    {attribute 'pytmc' := '
    pv: ACTUAL_POSISION;
    io: io;
    '}
    rActPosition : REAL;

    {attribute 'pytmc' := '
    pv: ACTUAL_ANGLE;
    io: io;
    '}
    rActAngle : REAL;



     {attribute 'pytmc' := '
    pv: HOME_READY;
    io: i;
    field: ZNAM False
    field: ONAM True
    '}
    bHomeReady:BOOL:=FALSE;


    //Local variables
    bInit: BOOL :=true;
    rTrig_Block: R_TRIG;
    rTrig_Open: R_TRIG;
    rTrig_Close: R_TRIG;

    //old values
    rOldReqPosition : REAL;
    rOldReqAngle: REAL;

    bExecuteMotionX: BOOL;


    fPosBlock: LREAL;
    fPosClose: LREAL;
    fPosOpen: LREAL;

    stSetPositionOptions: ST_SetPositionOptions;
    fbSetPosition_Pos: MC_SetPosition;
    fbSetPosition_Angle: MC_SetPosition;

    // For logging
    fbLogger : FB_LogMessage := (eSubsystem:=E_SubSystem.MOTION);
    tErrorPresent : R_TRIG;
    tAction : R_TRIG;
    tOverrideActivated : R_TRIG;

    FFO    :    FB_FastFault :=(
        i_DevName := 'OPT_XPM_Translation',
        i_Desc := 'Fault occurs when center is greated than that requested',
        i_TypeCode := 16#1010);


    bTest: BOOL;

    AptArrayStatus AT %Q* : ST_PMPS_Aperture_IO;
    AptArrayReq AT %I* : ST_PMPS_Aperture_IO;
END_VAR

// Initialize
ACT_init();

// Instantiate Function block for all the blades
ACT_Motion();

//SET and GET the requested and Actual values
ACT_CalculatePositions();

ACTION ACT_CalculatePositions:
//check if requested center or gap has changed
//check that the requested values are within acceptable motion range
IF (rOldReqPosition <> rReqPosition) THEN
        rOldReqPosition := rReqPosition;
        bExecuteMotionX := TRUE;
        fbLogger(sMsg:='Requested new Position.', eSevr:=TcEventSeverity.Verbose);
END_IF

IF (rOldReqAngle <> rReqAngle) THEN
    rOldReqAngle := rReqAngle;
    bExecuteMotionX := TRUE;
    fbLogger(sMsg:='Requested new Angle', eSevr:=TcEventSeverity.Verbose);
END_IF


//Calculate requested target positions from requested gap and center
fPosFirstStage		:= rReqPosition - rDistance / 2 * rReqAngle + rEncoderOffsetFirst;
fPosSecondStage		:= rReqPosition + rDistance / 2 * rReqAngle + rEncoderOffsetSecound;



//Calculate actual gap and center from actual stages positions
rActPosition	:= LREAL_TO_REAL( ((stFirstAxis.stAxisStatus.fActPosition - rEncoderOffsetFirst) + (stSecondAxis.stAxisStatus.fActPosition - rEncoderOffsetSecound)) / 2 );
rActAngle		:= LREAL_TO_REAL( ((stSecondAxis.stAxisStatus.fActPosition - rEncoderOffsetSecound) - (stFirstAxis.stAxisStatus.fActPosition - rEncoderOffsetFirst)) / rDistance );
END_ACTION

ACTION ACT_Init:

//  init the motion stages parameters
IF ( bInit) THEN
    stFirstAxis.bHardwareEnable := TRUE;
    stSecondAxis.bHardwareEnable := TRUE;
    stFirstAxis.bPowerSelf :=TRUE;
    stSecondAxis.bPowerSelf :=TRUE;
    stFirstAxis.nBrakeMode := ENUM_StageBrakeMode.NO_BRAKE;
    stSecondAxis.nBrakeMode := ENUM_StageBrakeMode.NO_BRAKE;
    FFO.i_DevName := i_DevName;
END_IF
END_ACTION

ACTION ACT_Motion:
// Instantiate Function block for all the blades
fbFirstStage(stMotionStage:=stFirstAxis);
fbSecondStage(stMotionStage:=stSecondAxis);



// PTP Motion for each blade
stFirst.sName := 'First';
stFirst.fPosition := fPosFirstStage;
stFirst.fDelta := fSmallDelta;
stFirst.fVelocity := fMaxVelocity;
stFirst.fAccel := fHighAccel;
stFirst.fDecel := fHighAccel;

stSecond.sName := 'Second';
stSecond.fPosition := fPosSecondStage;
stSecond.fDelta := fSmallDelta;
stSecond.fVelocity := fMaxVelocity;
stSecond.fAccel := fHighAccel;
stSecond.fDecel := fHighAccel;



IF (bExecuteMotionX) THEN
    fbFirst.bExecute := fbSecond.bExecute := bExecuteMotionX;
    bExecuteMotionX:= FALSE;
END_IF


fbFirst(
    stPositionState:=stFirst,
    bMoveOk:=bMoveOk,
    stMotionStage:=stFirstAxis);

fbSecond(
    stPositionState:=stSecond,
    bMoveOk:=bMoveOk,
    stMotionStage:=stSecondAxis);
END_ACTION

END_FUNCTION_BLOCK

// ---- POUs/PRG_OPT.TcPOU
PROGRAM PRG_OPT
VAR
	bInit: BOOL := TRUE;
	fbMotionRxG: FB_MotionStage;
	fbMotionXG: FB_MotionStage;
	fbMotionRzPM: FB_MotionStage;
END_VAR

IF bINIT THEN
	
	GVL_Main.M10.nBrakeMode := ENUM_StageBrakeMode.NO_BRAKE;
	GVL_Main.M10.bHardwareEnable := TRUE;
	GVL_Main.M10.bPowerSelf := TRUE;
	GVL_Main.M11.nBrakeMode := ENUM_StageBrakeMode.NO_BRAKE;
	GVL_Main.M11.bHardwareEnable := TRUE;
	GVL_Main.M11.bPowerSelf := TRUE;
	GVL_Main.M14.nBrakeMode := ENUM_StageBrakeMode.NO_BRAKE;
	GVL_Main.M14.bHardwareEnable := TRUE;
	GVL_Main.M14.bPowerSelf := TRUE;

	bINIT := FALSE;
END_IF;


fbMotionRxG(stMotionStage:= GVL_Main.M10);
fbMotionXG(stMotionStage:= GVL_Main.M11);
fbMotionRzPM(stMotionStage:= GVL_Main.M14);

END_PROGRAM

// ---- POUs/PRG_Sensor.TcPOU
PROGRAM PRG_Sensor
VAR
	bInit : bool :=TRUE;
	
    {attribute 'TcLinkTo' := 'TIIB[Rack#2D LinearGaugeAmp (SC-HG1-ETC)]^Process Data(Out) RxPDO-Map^Head Value Mode'}
	bSensorHeadValueMode AT %Q* : bool;
	
    {attribute 'TcLinkTo' := 'TIIB[Rack#2D LinearGaugeAmp (SC-HG1-ETC)]^Process Data(Out) RxPDO-Map^Normal Value Mode'}
	bSensorHeadNormalValueMode AT %Q* : bool;
	
	bResetSensorMode AT %I* : bool;
	
	uintTest AT %Q*: UINT;
	
END_VAR


If bInit Then
	bSensorHeadNormalValueMode := True;
	bInit := False;
End_If;

If(bResetSensorMode = True) Then
	bResetSensorMode := False;
	bSensorHeadValueMode := False;
	bSensorHeadNormalValueMode := False;
	bInit := True;
End_If;


GVL_Sensor.stYDF1.sName			:= 'YDF1 Panasonic HG-S';
GVL_Sensor.stYDF1.sEGU			:= 'mm';
GVL_Sensor.stYDF1.fCntsInEGU	:= 10000;
GVL_Sensor.stYDF2.sName			:= 'YDF2 Panasonic HG-S';
GVL_Sensor.stYDF2.sEGU			:= 'mm';
GVL_Sensor.stYDF2.fCntsInEGU	:= 10000;
GVL_Sensor.stYDF3.sName			:= 'YDF3 Panasonic HG-S';
GVL_Sensor.stYDF3.sEGU			:= 'mm';
GVL_Sensor.stYDF3.fCntsInEGU	:= 10000;
GVL_Sensor.stHDF.sName			:= 'HDF Panasonic HG-S';
GVL_Sensor.stHDF.sEGU			:= 'mm';
GVL_Sensor.stHDF.fCntsInEGU		:= 10000;

GVL_Sensor.stGraniteP.sName		:= 'Granite Pitch';
GVL_Sensor.stGraniteP.sEGU		:= 'mrad';
GVL_Sensor.stGraniteP.fCntsInEGU:= 3276.7; // 1V = 1mrad in Low gain mode
GVL_Sensor.stGraniteR.sName		:= 'Granite Roll';
GVL_Sensor.stGraniteR.sEGU		:= 'mrad';
GVL_Sensor.stGraniteR.fCntsInEGU:= 3276.7;

GVL_Sensor.stFrameP.sName		:= 'Det. Frame Pitch';
GVL_Sensor.stFrameP.sEGU		:= 'mrad';
GVL_Sensor.stFrameP.fCntsInEGU	:= 3276.7;
GVL_Sensor.stFrameR.sName		:= 'Det. Frame Roll';
GVL_Sensor.stFrameR.sEGU		:= 'mrad';
GVL_Sensor.stFrameR.fCntsInEGU	:= 3276.7;

GVL_Sensor.stPS1.sName			:= 'PS1';
GVL_Sensor.stPS1.sEGU			:= 'MPa';
GVL_Sensor.stPS1.fCntsInEGU		:= 13106.8;	// 0.25MPa/V
GVL_Sensor.stPS1.iOffset		:= 3277;	// 0MPa@1V  P=0.25(V-V0), V0 = 1.0

GVL_Sensor.stPS2.sName			:= 'PS2';
GVL_Sensor.stPS2.sEGU			:= 'MPa';
GVL_Sensor.stPS2.fCntsInEGU		:= 13106.8;	// 0.25MPa/V
GVL_Sensor.stPS2.iOffset		:= 3277;	// 0MPa@1V  P=0.25(V-V0), V0 = 1.0

GVL_Sensor.stPS3.sName			:= 'PS3';
GVL_Sensor.stPS3.sEGU			:= 'MPa';
GVL_Sensor.stPS3.fCntsInEGU		:= 13106.8;	// 0.25MPa/V
GVL_Sensor.stPS3.iOffset		:= 3277;	// 0MPa@1V  P=0.25(V-V0), V0 = 1.0

GVL_Sensor.stYDF1.fValue		:= DINT_TO_REAL(GVL_Sensor.stYDF1.iRawCnts - GVL_Sensor.stYDF1.iOffset) / GVL_Sensor.stYDF1.fCntsInEGU;
GVL_Sensor.stYDF2.fValue		:= DINT_TO_REAL(GVL_Sensor.stYDF2.iRawCnts - GVL_Sensor.stYDF2.iOffset) / GVL_Sensor.stYDF2.fCntsInEGU;
GVL_Sensor.stYDF3.fValue		:= DINT_TO_REAL(GVL_Sensor.stYDF3.iRawCnts - GVL_Sensor.stYDF3.iOffset) / GVL_Sensor.stYDF3.fCntsInEGU;
GVL_Sensor.stHDF.fValue			:= DINT_TO_REAL(GVL_Sensor.stHDF.iRawCnts  - GVL_Sensor.stHDF.iOffset)  / GVL_Sensor.stHDF.fCntsInEGU;
GVL_Sensor.stGraniteP.fValue	:= INT_TO_REAL(GVL_Sensor.stGraniteP.iRawCnts - GVL_Sensor.stGraniteP.iOffset) / GVL_Sensor.stGraniteP.fCntsInEGU;
GVL_Sensor.stGraniteR.fValue	:= INT_TO_REAL(GVL_Sensor.stGraniteR.iRawCnts - GVL_Sensor.stGraniteR.iOffset) / GVL_Sensor.stGraniteR.fCntsInEGU;
GVL_Sensor.stFrameP.fValue		:= INT_TO_REAL(GVL_Sensor.stFrameP.iRawCnts - GVL_Sensor.stFrameP.iOffset) / GVL_Sensor.stFrameP.fCntsInEGU;
GVL_Sensor.stFrameR.fValue		:= INT_TO_REAL(GVL_Sensor.stFrameR.iRawCnts - GVL_Sensor.stFrameR.iOffset) / GVL_Sensor.stFrameR.fCntsInEGU;

GVL_Sensor.stPS1.fValue			:= INT_TO_REAL(GVL_Sensor.stPS1.iRawCnts - GVL_Sensor.stPS1.iOffset) / GVL_Sensor.stPS1.fCntsInEGU;
GVL_Sensor.stPS2.fValue			:= INT_TO_REAL(GVL_Sensor.stPS2.iRawCnts - GVL_Sensor.stPS2.iOffset) / GVL_Sensor.stPS2.fCntsInEGU;
GVL_Sensor.stPS3.fValue			:= INT_TO_REAL(GVL_Sensor.stPS3.iRawCnts - GVL_Sensor.stPS3.iOffset) / GVL_Sensor.stPS3.fCntsInEGU;


//uintTest:= REAL_TO_UINT(GVL_Sensor.stYDF1.fValue);

END_PROGRAM
